LIN {X 0,Y 362.115,Z 224.377,A -85,B 0,C 180,E1 -12966.688,E2 -12966.688} C_VEL
LIN {X 0,Y 361.993,Z 224.393,A -85,B 0,C 180,E1 -12970.064,E2 -12970.064} C_VEL
LIN {X 0,Y 361.96,Z 224.393,A -85,B 0,C 180,E1 -12973.9,E2 -12973.9} C_VEL
LIN {X 0,Y 361.917,Z 224.398,A -85,B 0,C 180,E1 -12977.933,E2 -12977.933} C_VEL
LIN {X 0,Y 361.826,Z 224.413,A -85,B 0,C 180,E1 -12981.657,E2 -12981.657} C_VEL
LIN {X 0,Y 361.893,Z 224.405,A -85,B 0,C 180,E1 -12985.293,E2 -12985.293} C_VEL
LIN {X 0,Y 361.875,Z 224.406,A -85,B 0,C 180,E1 -12987.782,E2 -12987.782} C_VEL
LIN {X 0,Y 361.805,Z 224.415,A -85,B 0,C 180,E1 -12991.633,E2 -12991.633} C_VEL
LIN {X 0,Y 361.847,Z 224.405,A -85,B 0,C 180,E1 -12995.348,E2 -12995.348} C_VEL
LIN {X 0,Y 361.839,Z 224.413,A -85,B 0,C 180,E1 -12999.028,E2 -12999.028} C_VEL
LIN {X 0,Y 361.814,Z 224.411,A -85,B 0,C 180,E1 -13002.833,E2 -13002.833} C_VEL
LIN {X 0,Y 361.798,Z 224.416,A -85,B 0,C 180,E1 -13005.95,E2 -13005.95} C_VEL
LIN {X 0,Y 361.818,Z 224.414,A -85,B 0,C 180,E1 -13009.248,E2 -13009.248} C_VEL
LIN {X 0,Y 361.849,Z 224.412,A -85,B 0,C 180,E1 -13012.781,E2 -13012.781} C_VEL
LIN {X 0,Y 361.843,Z 224.414,A -85,B 0,C 180,E1 -13015.723,E2 -13015.723} C_VEL
LIN {X 0,Y 361.874,Z 224.521,A -85,B 0,C 180,E1 -13018.682,E2 -13018.682} C_VEL
LIN {X 0,Y 364.574,Z 235.414,A -85,B 0,C 180,E1 -13021.505,E2 -13021.505} C_VEL
LIN {X 0,Y 366.434,Z 244.952,A -85,B 0,C 180,E1 -13023.827,E2 -13023.827} C_VEL
LIN {X 0,Y 365.869,Z 253.146,A -85,B 0,C 180,E1 -13025.61,E2 -13025.61} C_VEL
LIN {X 0,Y 365.188,Z 259.855,A -85,B 0,C 180,E1 -13027.036,E2 -13027.036} C_VEL
LIN {X 0,Y 369.695,Z 284.03,A -85,B 0,C 180,E1 -13027.985,E2 -13027.985} C_VEL
LIN {X 0,Y 371.444,Z 298.142,A -85,B 0,C 180,E1 -13028.456,E2 -13028.456} C_VEL
LIN {X 0,Y 369.762,Z 370.004,A -85,B 0,C 180,E1 -13030.068,E2 -13030.068} C_VEL
LIN {X 0,Y 368.841,Z 384.089,A -85,B 0,C 180,E1 -13030.596,E2 -13030.596} C_VEL
LIN {X 0,Y 367.944,Z 396.187,A -85,B 0,C 180,E1 -13031.271,E2 -13031.271} C_VEL
LIN {X 0,Y 366.76,Z 407.982,A -85,B 0,C 180,E1 -13032.148,E2 -13032.148} C_VEL
LIN {X 0,Y 365.523,Z 419.416,A -85,B 0,C 180,E1 -13033.239,E2 -13033.239} C_VEL
LIN {X 0,Y 364.456,Z 428.714,A -85,B 0,C 180,E1 -13034.339,E2 -13034.339} C_VEL
LIN {X 0,Y 363.368,Z 438.309,A -85,B 0,C 180,E1 -13035.725,E2 -13035.725} C_VEL
LIN {X 0,Y 362.358,Z 447.58,A -85,B 0,C 180,E1 -13037.398,E2 -13037.398} C_VEL
LIN {X 0,Y 361.445,Z 455.08,A -85,B 0,C 180,E1 -13039.073,E2 -13039.073} C_VEL
LIN {X 0,Y 360.84,Z 461.992,A -85,B 0,C 180,E1 -13041.037,E2 -13041.037} C_VEL
LIN {X 0,Y 360.513,Z 466.581,A -85,B 0,C 180,E1 -13042.721,E2 -13042.721} C_VEL
LIN {X 0,Y 360.356,Z 470.071,A -85,B 0,C 180,E1 -13044.404,E2 -13044.404} C_VEL
LIN {X 0,Y 360.363,Z 471.821,A -85,B 0,C 180,E1 -13045.526,E2 -13045.526} C_VEL
LIN {X 0,Y 360.325,Z 473.156,A -85,B 0,C 180,E1 -13046.646,E2 -13046.646} C_VEL
LIN {X 0,Y 360.352,Z 474.073,A -85,B 0,C 180,E1 -13047.765,E2 -13047.765} C_VEL
LIN {X 0,Y 360.455,Z 474.543,A -85,B 0,C 180,E1 -13048.883,E2 -13048.883} C_VEL
LIN {X 0,Y 360.48,Z 474.608,A -85,B 0,C 180,E1 -13050,E2 -13050} C_VEL
LIN {X 0,Y 360.476,Z 474.272,A -85,B 0,C 180,E1 -13051.117,E2 -13051.117} C_VEL
LIN {X 0,Y 360.385,Z 473.507,A -85,B 0,C 180,E1 -13052.235,E2 -13052.235} C_VEL
LIN {X 0,Y 360.332,Z 472.287,A -85,B 0,C 180,E1 -13053.354,E2 -13053.354} C_VEL
LIN {X 0,Y 360.401,Z 469.667,A -85,B 0,C 180,E1 -13055.034,E2 -13055.034} C_VEL
LIN {X 0,Y 360.498,Z 465.984,A -85,B 0,C 180,E1 -13056.717,E2 -13056.717} C_VEL
LIN {X 0,Y 360.705,Z 461.141,A -85,B 0,C 180,E1 -13058.402,E2 -13058.402} C_VEL
LIN {X 0,Y 361.086,Z 454.997,A -85,B 0,C 180,E1 -13060.087,E2 -13060.087} C_VEL
LIN {X 0,Y 361.721,Z 447.337,A -85,B 0,C 180,E1 -13061.77,E2 -13061.77} C_VEL
LIN {X 0,Y 362.371,Z 439.494,A -85,B 0,C 180,E1 -13063.171,E2 -13063.171} C_VEL
LIN {X 0,Y 363.255,Z 429.911,A -85,B 0,C 180,E1 -13064.565,E2 -13064.565} C_VEL
LIN {X 0,Y 364.119,Z 419.27,A -85,B 0,C 180,E1 -13065.819,E2 -13065.819} C_VEL
LIN {X 0,Y 365.169,Z 407.451,A -85,B 0,C 180,E1 -13066.921,E2 -13066.921} C_VEL
LIN {X 0,Y 366.069,Z 394.843,A -85,B 0,C 180,E1 -13067.815,E2 -13067.815} C_VEL
LIN {X 0,Y 366.962,Z 381.699,A -85,B 0,C 180,E1 -13068.492,E2 -13068.492} C_VEL
LIN {X 0,Y 367.494,Z 368.498,A -85,B 0,C 180,E1 -13068.934,E2 -13068.934} C_VEL
LIN {X 0,Y 368.7,Z 295.929,A -85,B 0,C 180,E1 -13070.5,E2 -13070.5} C_VEL
LIN {X 0,Y 364.06,Z 262.327,A -85,B 0,C 180,E1 -13071.515,E2 -13071.515} C_VEL
LIN {X 0,Y 365.707,Z 244.487,A -85,B 0,C 180,E1 -13075.414,E2 -13075.414} C_VEL
LIN {X 0,Y 365.019,Z 239.454,A -85,B 0,C 180,E1 -13076.59,E2 -13076.59} C_VEL
LIN {X 0,Y 362.715,Z 228.266,A -85,B 0,C 180,E1 -13079.316,E2 -13079.316} C_VEL
LIN {X 0,Y 361.904,Z 224.406,A -85,B 0,C 180,E1 -13080.321,E2 -13080.321} C_VEL
LIN {X 0,Y 361.842,Z 224.412,A -85,B 0,C 180,E1 -13084.277,E2 -13084.277} C_VEL
LIN {X 0,Y 361.849,Z 224.409,A -85,B 0,C 180,E1 -13087.219,E2 -13087.219} C_VEL
LIN {X 0,Y 361.817,Z 224.412,A -85,B 0,C 180,E1 -13090.751,E2 -13090.751} C_VEL
LIN {X 0,Y 361.796,Z 224.416,A -85,B 0,C 180,E1 -13094.365,E2 -13094.365} C_VEL
LIN {X 0,Y 361.813,Z 224.417,A -85,B 0,C 180,E1 -13097.565,E2 -13097.565} C_VEL
LIN {X 0,Y 361.839,Z 224.41,A -85,B 0,C 180,E1 -13100.971,E2 -13100.971} C_VEL
LIN {X 0,Y 361.846,Z 224.408,A -85,B 0,C 180,E1 -13104.652,E2 -13104.652} C_VEL
LIN {X 0,Y 361.804,Z 224.414,A -85,B 0,C 180,E1 -13108.367,E2 -13108.367} C_VEL
LIN {X 0,Y 361.874,Z 224.405,A -85,B 0,C 180,E1 -13112.218,E2 -13112.218} C_VEL
LIN {X 0,Y 361.892,Z 224.403,A -85,B 0,C 180,E1 -13114.707,E2 -13114.707} C_VEL
LIN {X 0,Y 361.824,Z 224.411,A -85,B 0,C 180,E1 -13118.342,E2 -13118.342} C_VEL
LIN {X 0,Y 361.882,Z 224.404,A -85,B 0,C 180,E1 -13122.083,E2 -13122.083} C_VEL
LIN {X 0,Y 361.922,Z 224.404,A -85,B 0,C 180,E1 -13125.378,E2 -13125.378} C_VEL
LIN {X 0,Y 361.934,Z 224.4,A -85,B 0,C 180,E1 -13128.803,E2 -13128.803} C_VEL
LIN {X 0,Y 362.072,Z 224.38,A -85,B 0,C 180,E1 -13132.19,E2 -13132.19} C_VEL
LIN {X 0,Y 362.067,Z 224.382,A -85,B 0,C 180,E1 -13134.43,E2 -13134.43} C_VEL
LIN {X 0,Y 362.233,Z 224.36,A -85,B 0,C 180,E1 -13137.776,E2 -13137.776} C_VEL
LIN {X 0,Y 362.34,Z 224.347,A -85,B 0,C 180,E1 -13140,E2 -13140} C_VEL
LIN {X 0,Y 362.234,Z 224.361,A -85,B 0,C 180,E1 -13142.223,E2 -13142.223} C_VEL
LIN {X 0,Y 362.128,Z 224.378,A -85,B 0,C 180,E1 -13146.712,E2 -13146.712} C_VEL
LIN {X 0,Y 361.991,Z 224.391,A -85,B 0,C 180,E1 -13150.063,E2 -13150.063} C_VEL
LIN {X 0,Y 361.958,Z 224.395,A -85,B 0,C 180,E1 -13153.899,E2 -13153.899} C_VEL
LIN {X 0,Y 361.93,Z 224.399,A -85,B 0,C 180,E1 -13157.94,E2 -13157.94} C_VEL
LIN {X 0,Y 361.897,Z 224.402,A -85,B 0,C 180,E1 -13161.652,E2 -13161.652} C_VEL
LIN {X 0,Y 361.895,Z 224.402,A -85,B 0,C 180,E1 -13165.292,E2 -13165.292} C_VEL
LIN {X 0,Y 361.884,Z 224.405,A -85,B 0,C 180,E1 -13167.781,E2 -13167.781} C_VEL
LIN {X 0,Y 361.815,Z 224.412,A -85,B 0,C 180,E1 -13171.287,E2 -13171.287} C_VEL
LIN {X 0,Y 361.823,Z 224.418,A -85,B 0,C 180,E1 -13174.283,E2 -13174.283} C_VEL
LIN {X 0,Y 361.836,Z 224.41,A -85,B 0,C 180,E1 -13177.226,E2 -13177.226} C_VEL
LIN {X 0,Y 361.881,Z 224.405,A -85,B 0,C 180,E1 -13180.771,E2 -13180.771} C_VEL
LIN {X 0,Y 361.877,Z 224.408,A -85,B 0,C 180,E1 -13184.359,E2 -13184.359} C_VEL
LIN {X 0,Y 361.821,Z 224.413,A -85,B 0,C 180,E1 -13187.57,E2 -13187.57} C_VEL
LIN {X 0,Y 361.854,Z 224.407,A -85,B 0,C 180,E1 -13190.976,E2 -13190.976} C_VEL
LIN {X 0,Y 361.858,Z 224.407,A -85,B 0,C 180,E1 -13194.658,E2 -13194.658} C_VEL
LIN {X 0,Y 361.824,Z 224.412,A -85,B 0,C 180,E1 -13198.373,E2 -13198.373} C_VEL
LIN {X 0,Y 361.89,Z 224.403,A -85,B 0,C 180,E1 -13200.958,E2 -13200.958} C_VEL
LIN {X 0,Y 361.944,Z 224.4,A -85,B 0,C 180,E1 -13203.478,E2 -13203.478} C_VEL
LIN {X 0,Y 361.882,Z 224.406,A -85,B 0,C 180,E1 -13207.147,E2 -13207.147} C_VEL
LIN {X 0,Y 361.915,Z 224.4,A -85,B 0,C 180,E1 -13210.726,E2 -13210.726} C_VEL
LIN {X 0,Y 361.941,Z 224.397,A -85,B 0,C 180,E1 -13214.228,E2 -13214.228} C_VEL
LIN {X 0,Y 361.995,Z 224.39,A -85,B 0,C 180,E1 -13216.529,E2 -13216.529} C_VEL
LIN {X 0,Y 362.028,Z 224.387,A -85,B 0,C 180,E1 -13219.939,E2 -13219.939} C_VEL
LIN {X 0,Y 362.158,Z 224.376,A -85,B 0,C 180,E1 -13223.314,E2 -13223.314} C_VEL
LIN {X 0,Y 362.281,Z 224.356,A -85,B 0,C 180,E1 -13227.777,E2 -13227.777} C_VEL
LIN {X 0,Y 362.425,Z 224.337,A -85,B 0,C 180,E1 -13230,E2 -13230} C_VEL
LIN {X 0,Y 362.281,Z 224.354,A -85,B 0,C 180,E1 -13232.223,E2 -13232.223} C_VEL
LIN {X 0,Y 362.151,Z 224.373,A -85,B 0,C 180,E1 -13236.686,E2 -13236.686} C_VEL
LIN {X 0,Y 362.029,Z 224.386,A -85,B 0,C 180,E1 -13240.061,E2 -13240.061} C_VEL
LIN {X 0,Y 361.994,Z 224.39,A -85,B 0,C 180,E1 -13243.897,E2 -13243.897} C_VEL
LIN {X 0,Y 361.962,Z 224.394,A -85,B 0,C 180,E1 -13247.937,E2 -13247.937} C_VEL
LIN {X 0,Y 361.855,Z 224.407,A -85,B 0,C 180,E1 -13251.653,E2 -13251.653} C_VEL
LIN {X 0,Y 361.917,Z 224.405,A -85,B 0,C 180,E1 -13255.288,E2 -13255.288} C_VEL
LIN {X 0,Y 361.972,Z 224.536,A -85,B 0,C 180,E1 -13256.937,E2 -13256.937} C_VEL
LIN {X 0,Y 363.133,Z 230.494,A -85,B 0,C 180,E1 -13258.538,E2 -13258.538} C_VEL
LIN {X 0,Y 367.197,Z 242.914,A -85,B 0,C 180,E1 -13259.039,E2 -13259.039} C_VEL
LIN {X 0,Y 369.399,Z 254.487,A -85,B 0,C 180,E1 -13259.415,E2 -13259.415} C_VEL
LIN {X 0,Y 367.623,Z 338.548,A -85,B 0,C 180,E1 -13261.232,E2 -13261.232} C_VEL
LIN {X 0,Y 367.262,Z 348.263,A -85,B 0,C 180,E1 -13261.578,E2 -13261.578} C_VEL
LIN {X 0,Y 366.329,Z 353.922,A -85,B 0,C 180,E1 -13261.81,E2 -13261.81} C_VEL
LIN {X 0,Y 363.1,Z 362.978,A -85,B 0,C 180,E1 -13262.204,E2 -13262.204} C_VEL
LIN {X 0,Y 359.835,Z 371.762,A -85,B 0,C 180,E1 -13262.714,E2 -13262.714} C_VEL
LIN {X 0,Y 358.859,Z 376.971,A -85,B 0,C 180,E1 -13263.125,E2 -13263.125} C_VEL
LIN {X 0,Y 357.964,Z 387.984,A -85,B 0,C 180,E1 -13264.214,E2 -13264.214} C_VEL
LIN {X 0,Y 357.088,Z 398.297,A -85,B 0,C 180,E1 -13265.488,E2 -13265.488} C_VEL
LIN {X 0,Y 356.157,Z 408.096,A -85,B 0,C 180,E1 -13266.998,E2 -13266.998} C_VEL
LIN {X 0,Y 355.399,Z 416.152,A -85,B 0,C 180,E1 -13268.523,E2 -13268.523} C_VEL
LIN {X 0,Y 354.695,Z 423.012,A -85,B 0,C 180,E1 -13270.113,E2 -13270.113} C_VEL
LIN {X 0,Y 354.165,Z 428.666,A -85,B 0,C 180,E1 -13271.734,E2 -13271.734} C_VEL
LIN {X 0,Y 353.836,Z 433.362,A -85,B 0,C 180,E1 -13273.432,E2 -13273.432} C_VEL
LIN {X 0,Y 353.551,Z 436.816,A -85,B 0,C 180,E1 -13275.061,E2 -13275.061} C_VEL
LIN {X 0,Y 353.408,Z 438.217,A -85,B 0,C 180,E1 -13275.892,E2 -13275.892} C_VEL
LIN {X 0,Y 353.225,Z 440.195,A -85,B 0,C 180,E1 -13277.431,E2 -13277.431} C_VEL
LIN {X 0,Y 353.132,Z 441.501,A -85,B 0,C 180,E1 -13279.129,E2 -13279.129} C_VEL
LIN {X 0,Y 353.142,Z 441.899,A -85,B 0,C 180,E1 -13280.902,E2 -13280.902} C_VEL
LIN {X 0,Y 353.278,Z 441.286,A -85,B 0,C 180,E1 -13282.718,E2 -13282.718} C_VEL
LIN {X 0,Y 353.577,Z 439.303,A -85,B 0,C 180,E1 -13284.801,E2 -13284.801} C_VEL
LIN {X 0,Y 353.938,Z 436.632,A -85,B 0,C 180,E1 -13286.5,E2 -13286.5} C_VEL
LIN {X 0,Y 354.553,Z 432.301,A -85,B 0,C 180,E1 -13288.458,E2 -13288.458} C_VEL
LIN {X 0,Y 355.312,Z 426.61,A -85,B 0,C 180,E1 -13290.364,E2 -13290.364} C_VEL
LIN {X 0,Y 356.242,Z 419.66,A -85,B 0,C 180,E1 -13292.169,E2 -13292.169} C_VEL
LIN {X 0,Y 357.296,Z 412.146,A -85,B 0,C 180,E1 -13293.732,E2 -13293.732} C_VEL
LIN {X 0,Y 358.362,Z 403.424,A -85,B 0,C 180,E1 -13295.217,E2 -13295.217} C_VEL
LIN {X 0,Y 359.516,Z 393.604,A -85,B 0,C 180,E1 -13296.565,E2 -13296.565} C_VEL
LIN {X 0,Y 360.868,Z 381.992,A -85,B 0,C 180,E1 -13297.832,E2 -13297.832} C_VEL
LIN {X 0,Y 361.902,Z 370.101,A -85,B 0,C 180,E1 -13298.85,E2 -13298.85} C_VEL
LIN {X 0,Y 362.86,Z 357.252,A -85,B 0,C 180,E1 -13299.671,E2 -13299.671} C_VEL
LIN {X 0,Y 363.499,Z 344.303,A -85,B 0,C 180,E1 -13300.261,E2 -13300.261} C_VEL
LIN {X 0,Y 363.987,Z 329.813,A -85,B 0,C 180,E1 -13300.655,E2 -13300.655} C_VEL
LIN {X 0,Y 365.902,Z 256.319,A -85,B 0,C 180,E1 -13302.319,E2 -13302.319} C_VEL
LIN {X 0,Y 364.36,Z 250.049,A -85,B 0,C 180,E1 -13302.604,E2 -13302.604} C_VEL
LIN {X 0,Y 358.053,Z 235.223,A -85,B 0,C 180,E1 -13303.523,E2 -13303.523} C_VEL
LIN {X 0,Y 356.561,Z 231.883,A -85,B 0,C 180,E1 -13303.784,E2 -13303.784} C_VEL
LIN {X 0,Y 354.918,Z 225.281,A -85,B 0,C 180,E1 -13305.625,E2 -13305.625} C_VEL
LIN {X 0,Y 354.94,Z 225.278,A -85,B 0,C 180,E1 -13309.735,E2 -13309.735} C_VEL
LIN {X 0,Y 355.09,Z 225.255,A -85,B 0,C 180,E1 -13313.18,E2 -13313.18} C_VEL
LIN {X 0,Y 355.199,Z 225.241,A -85,B 0,C 180,E1 -13317.732,E2 -13317.732} C_VEL
LIN {X 0,Y 355.311,Z 225.226,A -85,B 0,C 180,E1 -13320,E2 -13320} C_VEL
LIN {X 0,Y 355.198,Z 225.24,A -85,B 0,C 180,E1 -13322.268,E2 -13322.268} C_VEL
LIN {X 0,Y 355.079,Z 225.255,A -85,B 0,C 180,E1 -13326.821,E2 -13326.821} C_VEL
LIN {X 0,Y 354.94,Z 225.272,A -85,B 0,C 180,E1 -13330.266,E2 -13330.266} C_VEL
LIN {X 0,Y 354.905,Z 225.272,A -85,B 0,C 180,E1 -13334.019,E2 -13334.019} C_VEL
LIN {X 0,Y 354.876,Z 225.276,A -85,B 0,C 180,E1 -13338.105,E2 -13338.105} C_VEL
LIN {X 0,Y 354.781,Z 225.292,A -85,B 0,C 180,E1 -13342.11,E2 -13342.11} C_VEL
LIN {X 0,Y 354.865,Z 225.28,A -85,B 0,C 180,E1 -13345.831,E2 -13345.831} C_VEL
LIN {X 0,Y 354.773,Z 225.286,A -85,B 0,C 180,E1 -13349.686,E2 -13349.686} C_VEL
LIN {X 0,Y 354.789,Z 225.289,A -85,B 0,C 180,E1 -13353.687,E2 -13353.687} C_VEL
LIN {X 0,Y 354.771,Z 225.294,A -85,B 0,C 180,E1 -13356.463,E2 -13356.463} C_VEL
LIN {X 0,Y 354.803,Z 225.289,A -85,B 0,C 180,E1 -13359.427,E2 -13359.427} C_VEL
LIN {X 0,Y 354.766,Z 225.289,A -85,B 0,C 180,E1 -13362.87,E2 -13362.87} C_VEL
LIN {X 0,Y 354.748,Z 225.295,A -85,B 0,C 180,E1 -13366.107,E2 -13366.107} C_VEL
LIN {X 0,Y 354.771,Z 225.292,A -85,B 0,C 180,E1 -13369.182,E2 -13369.182} C_VEL
LIN {X 0,Y 354.793,Z 225.293,A -85,B 0,C 180,E1 -13372.406,E2 -13372.406} C_VEL
LIN {X 0,Y 354.8,Z 225.288,A -85,B 0,C 180,E1 -13374.944,E2 -13374.944} C_VEL
LIN {X 0,Y 354.811,Z 225.417,A -85,B 0,C 180,E1 -13378.145,E2 -13378.145} C_VEL
LIN {X 0,Y 357.708,Z 236.939,A -85,B 0,C 180,E1 -13381.229,E2 -13381.229} C_VEL
LIN {X 0,Y 359.523,Z 246.075,A -85,B 0,C 180,E1 -13383.517,E2 -13383.517} C_VEL
LIN {X 0,Y 359.46,Z 250.516,A -85,B 0,C 180,E1 -13384.527,E2 -13384.527} C_VEL
LIN {X 0,Y 358.516,Z 259.669,A -85,B 0,C 180,E1 -13386.482,E2 -13386.482} C_VEL
LIN {X 0,Y 362.754,Z 281.64,A -85,B 0,C 180,E1 -13387.395,E2 -13387.395} C_VEL
LIN {X 0,Y 365.014,Z 298.796,A -85,B 0,C 180,E1 -13387.996,E2 -13387.996} C_VEL
LIN {X 0,Y 363.234,Z 369.682,A -85,B 0,C 180,E1 -13389.621,E2 -13389.621} C_VEL
LIN {X 0,Y 362.307,Z 383.682,A -85,B 0,C 180,E1 -13390.158,E2 -13390.158} C_VEL
LIN {X 0,Y 361.326,Z 395.747,A -85,B 0,C 180,E1 -13390.841,E2 -13390.841} C_VEL
LIN {X 0,Y 360.209,Z 406.735,A -85,B 0,C 180,E1 -13391.665,E2 -13391.665} C_VEL
LIN {X 0,Y 358.871,Z 418.31,A -85,B 0,C 180,E1 -13392.772,E2 -13392.772} C_VEL
LIN {X 0,Y 357.621,Z 428.82,A -85,B 0,C 180,E1 -13394.032,E2 -13394.032} C_VEL
LIN {X 0,Y 356.484,Z 438.319,A -85,B 0,C 180,E1 -13395.443,E2 -13395.443} C_VEL
LIN {X 0,Y 355.399,Z 447.532,A -85,B 0,C 180,E1 -13397.147,E2 -13397.147} C_VEL
LIN {X 0,Y 354.422,Z 454.987,A -85,B 0,C 180,E1 -13398.854,E2 -13398.854} C_VEL
LIN {X 0,Y 353.95,Z 460.048,A -85,B 0,C 180,E1 -13400.284,E2 -13400.284} C_VEL
LIN {X 0,Y 353.545,Z 464.985,A -85,B 0,C 180,E1 -13402.002,E2 -13402.002} C_VEL
LIN {X 0,Y 353.297,Z 469.445,A -85,B 0,C 180,E1 -13404.064,E2 -13404.064} C_VEL
LIN {X 0,Y 353.273,Z 471.556,A -85,B 0,C 180,E1 -13405.436,E2 -13405.436} C_VEL
LIN {X 0,Y 353.245,Z 472.878,A -85,B 0,C 180,E1 -13406.578,E2 -13406.578} C_VEL
LIN {X 0,Y 353.253,Z 473.765,A -85,B 0,C 180,E1 -13407.72,E2 -13407.72} C_VEL
LIN {X 0,Y 353.357,Z 474.218,A -85,B 0,C 180,E1 -13408.86,E2 -13408.86} C_VEL
LIN {X 0,Y 353.399,Z 474.269,A -85,B 0,C 180,E1 -13410,E2 -13410} C_VEL
LIN {X 0,Y 353.378,Z 473.915,A -85,B 0,C 180,E1 -13411.139,E2 -13411.139} C_VEL
LIN {X 0,Y 353.288,Z 473.116,A -85,B 0,C 180,E1 -13412.28,E2 -13412.28} C_VEL
LIN {X 0,Y 353.253,Z 471.879,A -85,B 0,C 180,E1 -13413.421,E2 -13413.421} C_VEL
LIN {X 0,Y 353.302,Z 469.218,A -85,B 0,C 180,E1 -13415.135,E2 -13415.135} C_VEL
LIN {X 0,Y 353.417,Z 465.492,A -85,B 0,C 180,E1 -13416.852,E2 -13416.852} C_VEL
LIN {X 0,Y 353.647,Z 460.602,A -85,B 0,C 180,E1 -13418.571,E2 -13418.571} C_VEL
LIN {X 0,Y 354.046,Z 454.404,A -85,B 0,C 180,E1 -13420.29,E2 -13420.29} C_VEL
LIN {X 0,Y 354.73,Z 446.681,A -85,B 0,C 180,E1 -13422.005,E2 -13422.005} C_VEL
LIN {X 0,Y 355.423,Z 438.753,A -85,B 0,C 180,E1 -13423.433,E2 -13423.433} C_VEL
LIN {X 0,Y 356.468,Z 428.191,A -85,B 0,C 180,E1 -13424.967,E2 -13424.967} C_VEL
LIN {X 0,Y 357.34,Z 416.984,A -85,B 0,C 180,E1 -13426.274,E2 -13426.274} C_VEL
LIN {X 0,Y 358.453,Z 404.493,A -85,B 0,C 180,E1 -13427.395,E2 -13427.395} C_VEL
LIN {X 0,Y 359.4,Z 392.315,A -85,B 0,C 180,E1 -13428.231,E2 -13428.231} C_VEL
LIN {X 0,Y 360.202,Z 378.807,A -85,B 0,C 180,E1 -13428.888,E2 -13428.888} C_VEL
LIN {X 0,Y 360.725,Z 365.466,A -85,B 0,C 180,E1 -13429.303,E2 -13429.303} C_VEL
LIN {X 0,Y 361.926,Z 296.685,A -85,B 0,C 180,E1 -13430.812,E2 -13430.812} C_VEL
LIN {X 0,Y 357.159,Z 262.03,A -85,B 0,C 180,E1 -13431.881,E2 -13431.881} C_VEL
LIN {X 0,Y 358.729,Z 245.661,A -85,B 0,C 180,E1 -13435.529,E2 -13435.529} C_VEL
LIN {X 0,Y 358.222,Z 241.554,A -85,B 0,C 180,E1 -13436.507,E2 -13436.507} C_VEL
LIN {X 0,Y 355.827,Z 229.809,A -85,B 0,C 180,E1 -13439.414,E2 -13439.414} C_VEL
LIN {X 0,Y 354.838,Z 225.285,A -85,B 0,C 180,E1 -13440.578,E2 -13440.578} C_VEL
LIN {X 0,Y 354.796,Z 225.29,A -85,B 0,C 180,E1 -13443.699,E2 -13443.699} C_VEL
LIN {X 0,Y 354.784,Z 225.29,A -85,B 0,C 180,E1 -13446.456,E2 -13446.456} C_VEL
LIN {X 0,Y 354.81,Z 225.287,A -85,B 0,C 180,E1 -13449.42,E2 -13449.42} C_VEL
LIN {X 0,Y 354.77,Z 225.29,A -85,B 0,C 180,E1 -13452.863,E2 -13452.863} C_VEL
LIN {X 0,Y 354.745,Z 225.296,A -85,B 0,C 180,E1 -13456.1,E2 -13456.1} C_VEL
LIN {X 0,Y 354.763,Z 225.292,A -85,B 0,C 180,E1 -13459.175,E2 -13459.175} C_VEL
LIN {X 0,Y 354.78,Z 225.289,A -85,B 0,C 180,E1 -13462.4,E2 -13462.4} C_VEL
LIN {X 0,Y 354.784,Z 225.289,A -85,B 0,C 180,E1 -13464.937,E2 -13464.937} C_VEL
LIN {X 0,Y 354.76,Z 225.291,A -85,B 0,C 180,E1 -13468.403,E2 -13468.403} C_VEL
LIN {X 0,Y 354.798,Z 225.291,A -85,B 0,C 180,E1 -13471.614,E2 -13471.614} C_VEL
LIN {X 0,Y 354.864,Z 225.279,A -85,B 0,C 180,E1 -13474.169,E2 -13474.169} C_VEL
LIN {X 0,Y 354.779,Z 225.29,A -85,B 0,C 180,E1 -13477.89,E2 -13477.89} C_VEL
LIN {X 0,Y 354.853,Z 225.28,A -85,B 0,C 180,E1 -13481.906,E2 -13481.906} C_VEL
LIN {X 0,Y 354.904,Z 225.273,A -85,B 0,C 180,E1 -13485.981,E2 -13485.981} C_VEL
LIN {X 0,Y 354.939,Z 225.27,A -85,B 0,C 180,E1 -13489.734,E2 -13489.734} C_VEL
LIN {X 0,Y 355.078,Z 225.257,A -85,B 0,C 180,E1 -13493.179,E2 -13493.179} C_VEL
LIN {X 0,Y 355.197,Z 225.237,A -85,B 0,C 180,E1 -13497.732,E2 -13497.732} C_VEL
LIN {X 0,Y 355.291,Z 225.225,A -85,B 0,C 180,E1 -13500,E2 -13500} C_VEL
LIN {X 0,Y 355.198,Z 225.237,A -85,B 0,C 180,E1 -13502.268,E2 -13502.268} C_VEL
LIN {X 0,Y 355.093,Z 225.256,A -85,B 0,C 180,E1 -13506.82,E2 -13506.82} C_VEL
LIN {X 0,Y 354.939,Z 225.271,A -85,B 0,C 180,E1 -13510.265,E2 -13510.265} C_VEL
LIN {X 0,Y 354.903,Z 225.274,A -85,B 0,C 180,E1 -13514.019,E2 -13514.019} C_VEL
LIN {X 0,Y 354.886,Z 225.277,A -85,B 0,C 180,E1 -13518.11,E2 -13518.11} C_VEL
LIN {X 0,Y 354.857,Z 225.281,A -85,B 0,C 180,E1 -13522.104,E2 -13522.104} C_VEL
LIN {X 0,Y 354.865,Z 225.279,A -85,B 0,C 180,E1 -13525.83,E2 -13525.83} C_VEL
LIN {X 0,Y 354.822,Z 225.284,A -85,B 0,C 180,E1 -13529.681,E2 -13529.681} C_VEL
LIN {X 0,Y 354.777,Z 225.29,A -85,B 0,C 180,E1 -13533.705,E2 -13533.705} C_VEL
LIN {X 0,Y 354.77,Z 225.294,A -85,B 0,C 180,E1 -13536.462,E2 -13536.462} C_VEL
LIN {X 0,Y 354.799,Z 225.287,A -85,B 0,C 180,E1 -13539.426,E2 -13539.426} C_VEL
LIN {X 0,Y 354.811,Z 225.285,A -85,B 0,C 180,E1 -13542.878,E2 -13542.878} C_VEL
LIN {X 0,Y 354.76,Z 225.297,A -85,B 0,C 180,E1 -13546.109,E2 -13546.109} C_VEL
LIN {X 0,Y 354.799,Z 225.286,A -85,B 0,C 180,E1 -13549.186,E2 -13549.186} C_VEL
LIN {X 0,Y 354.791,Z 225.289,A -85,B 0,C 180,E1 -13552.405,E2 -13552.405} C_VEL
LIN {X 0,Y 354.796,Z 225.287,A -85,B 0,C 180,E1 -13554.944,E2 -13554.944} C_VEL
LIN {X 0,Y 354.78,Z 225.29,A -85,B 0,C 180,E1 -13558.408,E2 -13558.408} C_VEL
LIN {X 0,Y 354.842,Z 225.286,A -85,B 0,C 180,E1 -13561.622,E2 -13561.622} C_VEL
LIN {X 0,Y 354.889,Z 225.277,A -85,B 0,C 180,E1 -13564.175,E2 -13564.175} C_VEL
LIN {X 0,Y 354.827,Z 225.286,A -85,B 0,C 180,E1 -13567.896,E2 -13567.896} C_VEL
LIN {X 0,Y 354.917,Z 225.274,A -85,B 0,C 180,E1 -13571.893,E2 -13571.893} C_VEL
LIN {X 0,Y 354.938,Z 225.27,A -85,B 0,C 180,E1 -13575.983,E2 -13575.983} C_VEL
LIN {X 0,Y 354.975,Z 225.267,A -85,B 0,C 180,E1 -13579.737,E2 -13579.737} C_VEL
LIN {X 0,Y 355.123,Z 225.251,A -85,B 0,C 180,E1 -13583.181,E2 -13583.181} C_VEL
LIN {X 0,Y 355.244,Z 225.233,A -85,B 0,C 180,E1 -13587.733,E2 -13587.733} C_VEL
LIN {X 0,Y 355.395,Z 225.212,A -85,B 0,C 180,E1 -13590,E2 -13590} C_VEL
LIN {X 0,Y 355.244,Z 225.231,A -85,B 0,C 180,E1 -13592.267,E2 -13592.267} C_VEL
LIN {X 0,Y 355.116,Z 225.25,A -85,B 0,C 180,E1 -13596.819,E2 -13596.819} C_VEL
LIN {X 0,Y 354.975,Z 225.265,A -85,B 0,C 180,E1 -13600.263,E2 -13600.263} C_VEL
LIN {X 0,Y 354.939,Z 225.269,A -85,B 0,C 180,E1 -13604.017,E2 -13604.017} C_VEL
LIN {X 0,Y 354.917,Z 225.272,A -85,B 0,C 180,E1 -13608.107,E2 -13608.107} C_VEL
LIN {X 0,Y 354.809,Z 225.286,A -85,B 0,C 180,E1 -13612.105,E2 -13612.105} C_VEL
LIN {X 0,Y 354.898,Z 225.278,A -85,B 0,C 180,E1 -13615.824,E2 -13615.824} C_VEL
LIN {X 0,Y 354.955,Z 225.341,A -85,B 0,C 180,E1 -13616.664,E2 -13616.664} C_VEL
LIN {X 0,Y 355.999,Z 230.651,A -85,B 0,C 180,E1 -13618.145,E2 -13618.145} C_VEL
LIN {X 0,Y 360.627,Z 244.841,A -85,B 0,C 180,E1 -13618.738,E2 -13618.738} C_VEL
LIN {X 0,Y 362.633,Z 256.13,A -85,B 0,C 180,E1 -13619.107,E2 -13619.107} C_VEL
LIN {X 0,Y 360.79,Z 339.016,A -85,B 0,C 180,E1 -13620.937,E2 -13620.937} C_VEL
LIN {X 0,Y 360.218,Z 352.523,A -85,B 0,C 180,E1 -13621.468,E2 -13621.468} C_VEL
LIN {X 0,Y 359.641,Z 365.466,A -85,B 0,C 180,E1 -13622.227,E2 -13622.227} C_VEL
LIN {X 0,Y 358.859,Z 376.971,A -85,B 0,C 180,E1 -13623.125,E2 -13623.125} C_VEL
LIN {X 0,Y 357.867,Z 382.128,A -85,B 0,C 180,E1 -13623.577,E2 -13623.577} C_VEL
LIN {X 0,Y 354.458,Z 390.195,A -85,B 0,C 180,E1 -13624.334,E2 -13624.334} C_VEL
LIN {X 0,Y 350.943,Z 397.796,A -85,B 0,C 180,E1 -13625.189,E2 -13625.189} C_VEL
LIN {X 0,Y 349.775,Z 402.191,A -85,B 0,C 180,E1 -13625.796,E2 -13625.796} C_VEL
LIN {X 0,Y 348.799,Z 411.724,A -85,B 0,C 180,E1 -13627.411,E2 -13627.411} C_VEL
LIN {X 0,Y 348.071,Z 419.314,A -85,B 0,C 180,E1 -13629,E2 -13629} C_VEL
LIN {X 0,Y 347.385,Z 426.608,A -85,B 0,C 180,E1 -13630.899,E2 -13630.899} C_VEL
LIN {X 0,Y 346.952,Z 431.555,A -85,B 0,C 180,E1 -13632.532,E2 -13632.532} C_VEL
LIN {X 0,Y 346.64,Z 435.473,A -85,B 0,C 180,E1 -13634.175,E2 -13634.175} C_VEL
LIN {X 0,Y 346.453,Z 437.499,A -85,B 0,C 180,E1 -13635.228,E2 -13635.228} C_VEL
LIN {X 0,Y 346.158,Z 440.007,A -85,B 0,C 180,E1 -13636.955,E2 -13636.955} C_VEL
LIN {X 0,Y 346.067,Z 441.58,A -85,B 0,C 180,E1 -13638.705,E2 -13638.705} C_VEL
LIN {X 0,Y 346.057,Z 442.237,A -85,B 0,C 180,E1 -13640.982,E2 -13640.982} C_VEL
LIN {X 0,Y 346.188,Z 441.846,A -85,B 0,C 180,E1 -13642.481,E2 -13642.481} C_VEL
LIN {X 0,Y 346.369,Z 440.489,A -85,B 0,C 180,E1 -13644.246,E2 -13644.246} C_VEL
LIN {X 0,Y 346.78,Z 437.897,A -85,B 0,C 180,E1 -13646.185,E2 -13646.185} C_VEL
LIN {X 0,Y 347.433,Z 433.678,A -85,B 0,C 180,E1 -13648.269,E2 -13648.269} C_VEL
LIN {X 0,Y 348.184,Z 428.332,A -85,B 0,C 180,E1 -13650.21,E2 -13650.21} C_VEL
LIN {X 0,Y 349.111,Z 421.757,A -85,B 0,C 180,E1 -13652.063,E2 -13652.063} C_VEL
LIN {X 0,Y 350.331,Z 413.84,A -85,B 0,C 180,E1 -13653.811,E2 -13653.811} C_VEL
LIN {X 0,Y 351.562,Z 404.378,A -85,B 0,C 180,E1 -13655.493,E2 -13655.493} C_VEL
LIN {X 0,Y 352.75,Z 394.91,A -85,B 0,C 180,E1 -13656.845,E2 -13656.845} C_VEL
LIN {X 0,Y 354.046,Z 384.237,A -85,B 0,C 180,E1 -13658.061,E2 -13658.061} C_VEL
LIN {X 0,Y 355.224,Z 372.344,A -85,B 0,C 180,E1 -13659.138,E2 -13659.138} C_VEL
LIN {X 0,Y 356.169,Z 360.62,A -85,B 0,C 180,E1 -13659.95,E2 -13659.95} C_VEL
LIN {X 0,Y 356.914,Z 347.135,A -85,B 0,C 180,E1 -13660.622,E2 -13660.622} C_VEL
LIN {X 0,Y 357.447,Z 334.632,A -85,B 0,C 180,E1 -13661.018,E2 -13661.018} C_VEL
LIN {X 0,Y 359.621,Z 257.658,A -85,B 0,C 180,E1 -13662.803,E2 -13662.803} C_VEL
LIN {X 0,Y 358.087,Z 252.005,A -85,B 0,C 180,E1 -13663.081,E2 -13663.081} C_VEL
LIN {X 0,Y 352.134,Z 238.191,A -85,B 0,C 180,E1 -13663.98,E2 -13663.98} C_VEL
LIN {X 0,Y 349.43,Z 232.448,A -85,B 0,C 180,E1 -13664.406,E2 -13664.406} C_VEL
LIN {X 0,Y 347.887,Z 226.158,A -85,B 0,C 180,E1 -13666.269,E2 -13666.269} C_VEL
LIN {X 0,Y 347.891,Z 226.158,A -85,B 0,C 180,E1 -13669.525,E2 -13669.525} C_VEL
LIN {X 0,Y 348.055,Z 226.131,A -85,B 0,C 180,E1 -13673.042,E2 -13673.042} C_VEL
LIN {X 0,Y 348.162,Z 226.118,A -85,B 0,C 180,E1 -13677.687,E2 -13677.687} C_VEL
LIN {X 0,Y 348.263,Z 226.104,A -85,B 0,C 180,E1 -13680,E2 -13680} C_VEL
LIN {X 0,Y 348.161,Z 226.117,A -85,B 0,C 180,E1 -13682.314,E2 -13682.314} C_VEL
LIN {X 0,Y 348.047,Z 226.132,A -85,B 0,C 180,E1 -13686.959,E2 -13686.959} C_VEL
LIN {X 0,Y 347.891,Z 226.151,A -85,B 0,C 180,E1 -13690.476,E2 -13690.476} C_VEL
LIN {X 0,Y 347.864,Z 226.149,A -85,B 0,C 180,E1 -13694.152,E2 -13694.152} C_VEL
LIN {X 0,Y 347.81,Z 226.157,A -85,B 0,C 180,E1 -13698.269,E2 -13698.269} C_VEL
LIN {X 0,Y 347.733,Z 226.169,A -85,B 0,C 180,E1 -13701.627,E2 -13701.627} C_VEL
LIN {X 0,Y 347.779,Z 226.164,A -85,B 0,C 180,E1 -13705.111,E2 -13705.111} C_VEL
LIN {X 0,Y 347.771,Z 226.162,A -85,B 0,C 180,E1 -13707.698,E2 -13707.698} C_VEL
LIN {X 0,Y 347.713,Z 226.171,A -85,B 0,C 180,E1 -13711.703,E2 -13711.703} C_VEL
LIN {X 0,Y 347.718,Z 226.171,A -85,B 0,C 180,E1 -13714.467,E2 -13714.467} C_VEL
LIN {X 0,Y 347.747,Z 226.166,A -85,B 0,C 180,E1 -13717.991,E2 -13717.991} C_VEL
LIN {X 0,Y 347.728,Z 226.17,A -85,B 0,C 180,E1 -13721.834,E2 -13721.834} C_VEL
LIN {X 0,Y 347.685,Z 226.172,A -85,B 0,C 180,E1 -13725.031,E2 -13725.031} C_VEL
LIN {X 0,Y 347.734,Z 226.171,A -85,B 0,C 180,E1 -13728.401,E2 -13728.401} C_VEL
LIN {X 0,Y 347.759,Z 226.166,A -85,B 0,C 180,E1 -13732.015,E2 -13732.015} C_VEL
LIN {X 0,Y 347.734,Z 226.17,A -85,B 0,C 180,E1 -13735.539,E2 -13735.539} C_VEL
LIN {X 0,Y 347.744,Z 226.255,A -85,B 0,C 180,E1 -13737.563,E2 -13737.563} C_VEL
LIN {X 0,Y 350.581,Z 237.158,A -85,B 0,C 180,E1 -13740.588,E2 -13740.588} C_VEL
LIN {X 0,Y 352.693,Z 247.677,A -85,B 0,C 180,E1 -13743.306,E2 -13743.306} C_VEL
LIN {X 0,Y 352.656,Z 252.007,A -85,B 0,C 180,E1 -13744.316,E2 -13744.316} C_VEL
LIN {X 0,Y 351.858,Z 259.022,A -85,B 0,C 180,E1 -13745.874,E2 -13745.874} C_VEL
LIN {X 0,Y 356.092,Z 280.965,A -85,B 0,C 180,E1 -13746.831,E2 -13746.831} C_VEL
LIN {X 0,Y 358.554,Z 298.254,A -85,B 0,C 180,E1 -13747.482,E2 -13747.482} C_VEL
LIN {X 0,Y 357.054,Z 357.395,A -85,B 0,C 180,E1 -13748.848,E2 -13748.848} C_VEL
LIN {X 0,Y 356.54,Z 373.684,A -85,B 0,C 180,E1 -13749.296,E2 -13749.296} C_VEL
LIN {X 0,Y 355.426,Z 387.387,A -85,B 0,C 180,E1 -13749.908,E2 -13749.908} C_VEL
LIN {X 0,Y 354.242,Z 400.349,A -85,B 0,C 180,E1 -13750.744,E2 -13750.744} C_VEL
LIN {X 0,Y 352.952,Z 411.807,A -85,B 0,C 180,E1 -13751.725,E2 -13751.725} C_VEL
LIN {X 0,Y 351.488,Z 423.483,A -85,B 0,C 180,E1 -13752.999,E2 -13752.999} C_VEL
LIN {X 0,Y 350.177,Z 433.966,A -85,B 0,C 180,E1 -13754.442,E2 -13754.442} C_VEL
LIN {X 0,Y 349.024,Z 443.147,A -85,B 0,C 180,E1 -13756.019,E2 -13756.019} C_VEL
LIN {X 0,Y 347.902,Z 451.389,A -85,B 0,C 180,E1 -13757.755,E2 -13757.755} C_VEL
LIN {X 0,Y 347.147,Z 458.033,A -85,B 0,C 180,E1 -13759.503,E2 -13759.503} C_VEL
LIN {X 0,Y 346.629,Z 463.327,A -85,B 0,C 180,E1 -13761.254,E2 -13761.254} C_VEL
LIN {X 0,Y 346.322,Z 467.456,A -85,B 0,C 180,E1 -13763.007,E2 -13763.007} C_VEL
LIN {X 0,Y 346.202,Z 469.592,A -85,B 0,C 180,E1 -13764.175,E2 -13764.175} C_VEL
LIN {X 0,Y 346.169,Z 471.306,A -85,B 0,C 180,E1 -13765.342,E2 -13765.342} C_VEL
LIN {X 0,Y 346.166,Z 472.609,A -85,B 0,C 180,E1 -13766.508,E2 -13766.508} C_VEL
LIN {X 0,Y 346.159,Z 473.458,A -85,B 0,C 180,E1 -13767.673,E2 -13767.673} C_VEL
LIN {X 0,Y 346.259,Z 473.894,A -85,B 0,C 180,E1 -13768.837,E2 -13768.837} C_VEL
LIN {X 0,Y 346.32,Z 473.929,A -85,B 0,C 180,E1 -13770,E2 -13770} C_VEL
LIN {X 0,Y 346.281,Z 473.555,A -85,B 0,C 180,E1 -13771.163,E2 -13771.163} C_VEL
LIN {X 0,Y 346.191,Z 472.722,A -85,B 0,C 180,E1 -13772.327,E2 -13772.327} C_VEL
LIN {X 0,Y 346.176,Z 471.468,A -85,B 0,C 180,E1 -13773.491,E2 -13773.491} C_VEL
LIN {X 0,Y 346.21,Z 468.767,A -85,B 0,C 180,E1 -13775.241,E2 -13775.241} C_VEL
LIN {X 0,Y 346.341,Z 464.998,A -85,B 0,C 180,E1 -13776.992,E2 -13776.992} C_VEL
LIN {X 0,Y 346.571,Z 460.059,A -85,B 0,C 180,E1 -13778.747,E2 -13778.747} C_VEL
LIN {X 0,Y 346.988,Z 453.805,A -85,B 0,C 180,E1 -13780.502,E2 -13780.502} C_VEL
LIN {X 0,Y 347.723,Z 446.003,A -85,B 0,C 180,E1 -13782.251,E2 -13782.251} C_VEL
LIN {X 0,Y 348.494,Z 437.986,A -85,B 0,C 180,E1 -13783.706,E2 -13783.706} C_VEL
LIN {X 0,Y 349.459,Z 428.199,A -85,B 0,C 180,E1 -13785.154,E2 -13785.154} C_VEL
LIN {X 0,Y 350.349,Z 417.321,A -85,B 0,C 180,E1 -13786.458,E2 -13786.458} C_VEL
LIN {X 0,Y 351.385,Z 406.806,A -85,B 0,C 180,E1 -13787.456,E2 -13787.456} C_VEL
LIN {X 0,Y 352.353,Z 394.202,A -85,B 0,C 180,E1 -13788.382,E2 -13788.382} C_VEL
LIN {X 0,Y 353.27,Z 381.072,A -85,B 0,C 180,E1 -13789.085,E2 -13789.085} C_VEL
LIN {X 0,Y 353.824,Z 367.93,A -85,B 0,C 180,E1 -13789.544,E2 -13789.544} C_VEL
LIN {X 0,Y 355.188,Z 297.497,A -85,B 0,C 180,E1 -13791.132,E2 -13791.132} C_VEL
LIN {X 0,Y 350.249,Z 261.768,A -85,B 0,C 180,E1 -13792.251,E2 -13792.251} C_VEL
LIN {X 0,Y 351.791,Z 246.207,A -85,B 0,C 180,E1 -13795.792,E2 -13795.792} C_VEL
LIN {X 0,Y 349.716,Z 234.961,A -85,B 0,C 180,E1 -13798.589,E2 -13798.589} C_VEL
LIN {X 0,Y 347.782,Z 226.164,A -85,B 0,C 180,E1 -13800.887,E2 -13800.887} C_VEL
LIN {X 0,Y 347.733,Z 226.168,A -85,B 0,C 180,E1 -13804.461,E2 -13804.461} C_VEL
LIN {X 0,Y 347.759,Z 226.169,A -85,B 0,C 180,E1 -13807.985,E2 -13807.985} C_VEL
LIN {X 0,Y 347.733,Z 226.172,A -85,B 0,C 180,E1 -13811.827,E2 -13811.827} C_VEL
LIN {X 0,Y 347.684,Z 226.173,A -85,B 0,C 180,E1 -13815.024,E2 -13815.024} C_VEL
LIN {X 0,Y 347.728,Z 226.168,A -85,B 0,C 180,E1 -13818.394,E2 -13818.394} C_VEL
LIN {X 0,Y 347.746,Z 226.167,A -85,B 0,C 180,E1 -13822.009,E2 -13822.009} C_VEL
LIN {X 0,Y 347.717,Z 226.174,A -85,B 0,C 180,E1 -13825.533,E2 -13825.533} C_VEL
LIN {X 0,Y 347.712,Z 226.169,A -85,B 0,C 180,E1 -13828.297,E2 -13828.297} C_VEL
LIN {X 0,Y 347.77,Z 226.162,A -85,B 0,C 180,E1 -13832.302,E2 -13832.302} C_VEL
LIN {X 0,Y 347.783,Z 226.167,A -85,B 0,C 180,E1 -13835.403,E2 -13835.403} C_VEL
LIN {X 0,Y 347.744,Z 226.166,A -85,B 0,C 180,E1 -13838.667,E2 -13838.667} C_VEL
LIN {X 0,Y 347.805,Z 226.158,A -85,B 0,C 180,E1 -13842.356,E2 -13842.356} C_VEL
LIN {X 0,Y 347.862,Z 226.151,A -85,B 0,C 180,E1 -13845.969,E2 -13845.969} C_VEL
LIN {X 0,Y 347.89,Z 226.149,A -85,B 0,C 180,E1 -13849.524,E2 -13849.524} C_VEL
LIN {X 0,Y 348.046,Z 226.134,A -85,B 0,C 180,E1 -13853.041,E2 -13853.041} C_VEL
LIN {X 0,Y 348.16,Z 226.114,A -85,B 0,C 180,E1 -13857.686,E2 -13857.686} C_VEL
LIN {X 0,Y 348.243,Z 226.103,A -85,B 0,C 180,E1 -13860,E2 -13860} C_VEL
LIN {X 0,Y 348.161,Z 226.114,A -85,B 0,C 180,E1 -13862.313,E2 -13862.313} C_VEL
LIN {X 0,Y 348.058,Z 226.131,A -85,B 0,C 180,E1 -13866.958,E2 -13866.958} C_VEL
LIN {X 0,Y 347.89,Z 226.15,A -85,B 0,C 180,E1 -13870.475,E2 -13870.475} C_VEL
LIN {X 0,Y 347.862,Z 226.152,A -85,B 0,C 180,E1 -13874.151,E2 -13874.151} C_VEL
LIN {X 0,Y 347.855,Z 226.154,A -85,B 0,C 180,E1 -13878.292,E2 -13878.292} C_VEL
LIN {X 0,Y 347.805,Z 226.158,A -85,B 0,C 180,E1 -13881.658,E2 -13881.658} C_VEL
LIN {X 0,Y 347.786,Z 226.161,A -85,B 0,C 180,E1 -13885.11,E2 -13885.11} C_VEL
LIN {X 0,Y 347.778,Z 226.161,A -85,B 0,C 180,E1 -13887.696,E2 -13887.696} C_VEL
LIN {X 0,Y 347.732,Z 226.173,A -85,B 0,C 180,E1 -13890.349,E2 -13890.349} C_VEL
LIN {X 0,Y 347.715,Z 226.173,A -85,B 0,C 180,E1 -13894.467,E2 -13894.467} C_VEL
LIN {X 0,Y 347.748,Z 226.169,A -85,B 0,C 180,E1 -13897.991,E2 -13897.991} C_VEL
LIN {X 0,Y 347.761,Z 226.164,A -85,B 0,C 180,E1 -13901.612,E2 -13901.612} C_VEL
LIN {X 0,Y 347.752,Z 226.164,A -85,B 0,C 180,E1 -13905.018,E2 -13905.018} C_VEL
LIN {X 0,Y 347.742,Z 226.168,A -85,B 0,C 180,E1 -13908.398,E2 -13908.398} C_VEL
LIN {X 0,Y 347.757,Z 226.169,A -85,B 0,C 180,E1 -13912.014,E2 -13912.014} C_VEL
LIN {X 0,Y 347.729,Z 226.17,A -85,B 0,C 180,E1 -13915.539,E2 -13915.539} C_VEL
LIN {X 0,Y 347.752,Z 226.169,A -85,B 0,C 180,E1 -13919.656,E2 -13919.656} C_VEL
LIN {X 0,Y 347.842,Z 226.153,A -85,B 0,C 180,E1 -13922.747,E2 -13922.747} C_VEL
LIN {X 0,Y 347.78,Z 226.162,A -85,B 0,C 180,E1 -13926.164,E2 -13926.164} C_VEL
LIN {X 0,Y 347.811,Z 226.16,A -85,B 0,C 180,E1 -13929.912,E2 -13929.912} C_VEL
LIN {X 0,Y 347.861,Z 226.151,A -85,B 0,C 180,E1 -13932.361,E2 -13932.361} C_VEL
LIN {X 0,Y 347.893,Z 226.148,A -85,B 0,C 180,E1 -13935.972,E2 -13935.972} C_VEL
LIN {X 0,Y 347.925,Z 226.147,A -85,B 0,C 180,E1 -13939.527,E2 -13939.527} C_VEL
LIN {X 0,Y 348.089,Z 226.125,A -85,B 0,C 180,E1 -13943.043,E2 -13943.043} C_VEL
LIN {X 0,Y 348.206,Z 226.11,A -85,B 0,C 180,E1 -13947.687,E2 -13947.687} C_VEL
LIN {X 0,Y 348.343,Z 226.091,A -85,B 0,C 180,E1 -13950,E2 -13950} C_VEL
LIN {X 0,Y 348.207,Z 226.108,A -85,B 0,C 180,E1 -13952.313,E2 -13952.313} C_VEL
LIN {X 0,Y 348.083,Z 226.128,A -85,B 0,C 180,E1 -13956.957,E2 -13956.957} C_VEL
LIN {X 0,Y 347.926,Z 226.144,A -85,B 0,C 180,E1 -13960.473,E2 -13960.473} C_VEL
LIN {X 0,Y 347.895,Z 226.147,A -85,B 0,C 180,E1 -13964.149,E2 -13964.149} C_VEL
LIN {X 0,Y 347.885,Z 226.149,A -85,B 0,C 180,E1 -13968.288,E2 -13968.288} C_VEL
LIN {X 0,Y 347.761,Z 226.163,A -85,B 0,C 180,E1 -13971.624,E2 -13971.624} C_VEL
LIN {X 0,Y 347.806,Z 226.163,A -85,B 0,C 180,E1 -13975.106,E2 -13975.106} C_VEL
LIN {X 0,Y 347.891,Z 226.263,A -85,B 0,C 180,E1 -13976.418,E2 -13976.418} C_VEL
LIN {X 0,Y 348.836,Z 231.046,A -85,B 0,C 180,E1 -13977.767,E2 -13977.767} C_VEL
LIN {X 0,Y 354.108,Z 247.007,A -85,B 0,C 180,E1 -13978.443,E2 -13978.443} C_VEL
LIN {X 0,Y 355.88,Z 256.822,A -85,B 0,C 180,E1 -13978.772,E2 -13978.772} C_VEL
LIN {X 0,Y 353.995,Z 338.747,A -85,B 0,C 180,E1 -13980.618,E2 -13980.618} C_VEL
LIN {X 0,Y 353.388,Z 352.346,A -85,B 0,C 180,E1 -13981.154,E2 -13981.154} C_VEL
LIN {X 0,Y 352.839,Z 364.787,A -85,B 0,C 180,E1 -13981.881,E2 -13981.881} C_VEL
LIN {X 0,Y 352.015,Z 376.432,A -85,B 0,C 180,E1 -13982.788,E2 -13982.788} C_VEL
LIN {X 0,Y 351.059,Z 388.057,A -85,B 0,C 180,E1 -13983.95,E2 -13983.95} C_VEL
LIN {X 0,Y 350.232,Z 397.514,A -85,B 0,C 180,E1 -13985.124,E2 -13985.124} C_VEL
LIN {X 0,Y 349.775,Z 402.191,A -85,B 0,C 180,E1 -13985.796,E2 -13985.796} C_VEL
LIN {X 0,Y 348.627,Z 406.494,A -85,B 0,C 180,E1 -13986.436,E2 -13986.436} C_VEL
LIN {X 0,Y 345.145,Z 413.068,A -85,B 0,C 180,E1 -13987.522,E2 -13987.522} C_VEL
LIN {X 0,Y 341.744,Z 419.021,A -85,B 0,C 180,E1 -13988.718,E2 -13988.718} C_VEL
LIN {X 0,Y 340.737,Z 422.35,A -85,B 0,C 180,E1 -13989.522,E2 -13989.522} C_VEL
LIN {X 0,Y 340.096,Z 428.827,A -85,B 0,C 180,E1 -13991.391,E2 -13991.391} C_VEL
LIN {X 0,Y 339.725,Z 433.358,A -85,B 0,C 180,E1 -13993.048,E2 -13993.048} C_VEL
LIN {X 0,Y 339.422,Z 436.977,A -85,B 0,C 180,E1 -13994.742,E2 -13994.742} C_VEL
LIN {X 0,Y 339.089,Z 440.184,A -85,B 0,C 180,E1 -13996.847,E2 -13996.847} C_VEL
LIN {X 0,Y 338.993,Z 441.685,A -85,B 0,C 180,E1 -13998.439,E2 -13998.439} C_VEL
LIN {X 0,Y 338.963,Z 442.479,A -85,B 0,C 180,E1 -14000.091,E2 -14000.091} C_VEL
LIN {X 0,Y 339.016,Z 442.421,A -85,B 0,C 180,E1 -14001.969,E2 -14001.969} C_VEL
LIN {X 0,Y 339.241,Z 441.301,A -85,B 0,C 180,E1 -14003.888,E2 -14003.888} C_VEL
LIN {X 0,Y 339.684,Z 438.751,A -85,B 0,C 180,E1 -14006.04,E2 -14006.04} C_VEL
LIN {X 0,Y 340.225,Z 435.453,A -85,B 0,C 180,E1 -14007.87,E2 -14007.87} C_VEL
LIN {X 0,Y 340.997,Z 430.353,A -85,B 0,C 180,E1 -14009.944,E2 -14009.944} C_VEL
LIN {X 0,Y 341.925,Z 424.359,A -85,B 0,C 180,E1 -14011.788,E2 -14011.788} C_VEL
LIN {X 0,Y 343.215,Z 416.246,A -85,B 0,C 180,E1 -14013.745,E2 -14013.745} C_VEL
LIN {X 0,Y 344.362,Z 408.384,A -85,B 0,C 180,E1 -14015.268,E2 -14015.268} C_VEL
LIN {X 0,Y 345.682,Z 398.205,A -85,B 0,C 180,E1 -14016.858,E2 -14016.858} C_VEL
LIN {X 0,Y 347.055,Z 387.765,A -85,B 0,C 180,E1 -14018.155,E2 -14018.155} C_VEL
LIN {X 0,Y 348.216,Z 377.688,A -85,B 0,C 180,E1 -14019.163,E2 -14019.163} C_VEL
LIN {X 0,Y 349.282,Z 365.908,A -85,B 0,C 180,E1 -14020.099,E2 -14020.099} C_VEL
LIN {X 0,Y 350.225,Z 352.29,A -85,B 0,C 180,E1 -14020.892,E2 -14020.892} C_VEL
LIN {X 0,Y 350.825,Z 339.439,A -85,B 0,C 180,E1 -14021.396,E2 -14021.396} C_VEL
LIN {X 0,Y 353.34,Z 258.911,A -85,B 0,C 180,E1 -14023.312,E2 -14023.312} C_VEL
LIN {X 0,Y 352.111,Z 254.744,A -85,B 0,C 180,E1 -14023.532,E2 -14023.532} C_VEL
LIN {X 0,Y 345.589,Z 239.584,A -85,B 0,C 180,E1 -14024.566,E2 -14024.566} C_VEL
LIN {X 0,Y 342.331,Z 232.842,A -85,B 0,C 180,E1 -14025.104,E2 -14025.104} C_VEL
LIN {X 0,Y 340.823,Z 227.038,A -85,B 0,C 180,E1 -14026.89,E2 -14026.89} C_VEL
LIN {X 0,Y 340.876,Z 227.028,A -85,B 0,C 180,E1 -14030.507,E2 -14030.507} C_VEL
LIN {X 0,Y 341.023,Z 227.008,A -85,B 0,C 180,E1 -14032.898,E2 -14032.898} C_VEL
LIN {X 0,Y 341.124,Z 226.995,A -85,B 0,C 180,E1 -14037.639,E2 -14037.639} C_VEL
LIN {X 0,Y 341.214,Z 226.982,A -85,B 0,C 180,E1 -14040,E2 -14040} C_VEL
LIN {X 0,Y 341.123,Z 226.994,A -85,B 0,C 180,E1 -14042.362,E2 -14042.362} C_VEL
LIN {X 0,Y 341.016,Z 227.009,A -85,B 0,C 180,E1 -14047.103,E2 -14047.103} C_VEL
LIN {X 0,Y 340.834,Z 227.028,A -85,B 0,C 180,E1 -14050.695,E2 -14050.695} C_VEL
LIN {X 0,Y 340.829,Z 227.025,A -85,B 0,C 180,E1 -14054.327,E2 -14054.327} C_VEL
LIN {X 0,Y 340.763,Z 227.037,A -85,B 0,C 180,E1 -14058.448,E2 -14058.448} C_VEL
LIN {X 0,Y 340.687,Z 227.047,A -85,B 0,C 180,E1 -14061.844,E2 -14061.844} C_VEL
LIN {X 0,Y 340.74,Z 227.039,A -85,B 0,C 180,E1 -14065.667,E2 -14065.667} C_VEL
LIN {X 0,Y 340.689,Z 227.048,A -85,B 0,C 180,E1 -14068.325,E2 -14068.325} C_VEL
LIN {X 0,Y 340.664,Z 227.05,A -85,B 0,C 180,E1 -14071.049,E2 -14071.049} C_VEL
LIN {X 0,Y 340.692,Z 227.041,A -85,B 0,C 180,E1 -14075.282,E2 -14075.282} C_VEL
LIN {X 0,Y 340.685,Z 227.045,A -85,B 0,C 180,E1 -14078.389,E2 -14078.389} C_VEL
LIN {X 0,Y 340.677,Z 227.05,A -85,B 0,C 180,E1 -14082.048,E2 -14082.048} C_VEL
LIN {X 0,Y 340.634,Z 227.054,A -85,B 0,C 180,E1 -14086.231,E2 -14086.231} C_VEL
LIN {X 0,Y 340.672,Z 227.047,A -85,B 0,C 180,E1 -14089.757,E2 -14089.757} C_VEL
LIN {X 0,Y 340.692,Z 227.046,A -85,B 0,C 180,E1 -14093.261,E2 -14093.261} C_VEL
LIN {X 0,Y 340.703,Z 227.177,A -85,B 0,C 180,E1 -14096.956,E2 -14096.956} C_VEL
LIN {X 0,Y 343.783,Z 238.903,A -85,B 0,C 180,E1 -14100.326,E2 -14100.326} C_VEL
LIN {X 0,Y 345.906,Z 249.487,A -85,B 0,C 180,E1 -14103.127,E2 -14103.127} C_VEL
LIN {X 0,Y 345.872,Z 253.547,A -85,B 0,C 180,E1 -14104.099,E2 -14104.099} C_VEL
LIN {X 0,Y 345.291,Z 258.561,A -85,B 0,C 180,E1 -14105.241,E2 -14105.241} C_VEL
LIN {X 0,Y 349.782,Z 281.783,A -85,B 0,C 180,E1 -14106.309,E2 -14106.309} C_VEL
LIN {X 0,Y 352.28,Z 299.59,A -85,B 0,C 180,E1 -14106.996,E2 -14106.996} C_VEL
LIN {X 0,Y 350.306,Z 369.294,A -85,B 0,C 180,E1 -14108.679,E2 -14108.679} C_VEL
LIN {X 0,Y 349.301,Z 383.125,A -85,B 0,C 180,E1 -14109.232,E2 -14109.232} C_VEL
LIN {X 0,Y 348.215,Z 395.136,A -85,B 0,C 180,E1 -14109.936,E2 -14109.936} C_VEL
LIN {X 0,Y 346.831,Z 407.673,A -85,B 0,C 180,E1 -14110.931,E2 -14110.931} C_VEL
LIN {X 0,Y 345.35,Z 418.948,A -85,B 0,C 180,E1 -14112.075,E2 -14112.075} C_VEL
LIN {X 0,Y 343.978,Z 429.175,A -85,B 0,C 180,E1 -14113.381,E2 -14113.381} C_VEL
LIN {X 0,Y 342.754,Z 438.43,A -85,B 0,C 180,E1 -14114.847,E2 -14114.847} C_VEL
LIN {X 0,Y 341.52,Z 447.496,A -85,B 0,C 180,E1 -14116.615,E2 -14116.615} C_VEL
LIN {X 0,Y 340.442,Z 454.818,A -85,B 0,C 180,E1 -14118.39,E2 -14118.39} C_VEL
LIN {X 0,Y 339.916,Z 459.785,A -85,B 0,C 180,E1 -14119.879,E2 -14119.879} C_VEL
LIN {X 0,Y 339.438,Z 464.639,A -85,B 0,C 180,E1 -14121.667,E2 -14121.667} C_VEL
LIN {X 0,Y 339.164,Z 468.365,A -85,B 0,C 180,E1 -14123.456,E2 -14123.456} C_VEL
LIN {X 0,Y 339.071,Z 471.059,A -85,B 0,C 180,E1 -14125.245,E2 -14125.245} C_VEL
LIN {X 0,Y 339.088,Z 472.336,A -85,B 0,C 180,E1 -14126.435,E2 -14126.435} C_VEL
LIN {X 0,Y 339.16,Z 473.57,A -85,B 0,C 180,E1 -14128.813,E2 -14128.813} C_VEL
LIN {X 0,Y 339.227,Z 473.586,A -85,B 0,C 180,E1 -14130,E2 -14130} C_VEL
LIN {X 0,Y 339.185,Z 473.181,A -85,B 0,C 180,E1 -14131.187,E2 -14131.187} C_VEL
LIN {X 0,Y 339.098,Z 472.315,A -85,B 0,C 180,E1 -14132.375,E2 -14132.375} C_VEL
LIN {X 0,Y 339.101,Z 471.04,A -85,B 0,C 180,E1 -14133.564,E2 -14133.564} C_VEL
LIN {X 0,Y 339.127,Z 468.056,A -85,B 0,C 180,E1 -14135.479,E2 -14135.479} C_VEL
LIN {X 0,Y 339.268,Z 464.469,A -85,B 0,C 180,E1 -14137.139,E2 -14137.139} C_VEL
LIN {X 0,Y 339.516,Z 459.473,A -85,B 0,C 180,E1 -14138.93,E2 -14138.93} C_VEL
LIN {X 0,Y 339.938,Z 453.151,A -85,B 0,C 180,E1 -14140.722,E2 -14140.722} C_VEL
LIN {X 0,Y 340.746,Z 445.243,A -85,B 0,C 180,E1 -14142.506,E2 -14142.506} C_VEL
LIN {X 0,Y 341.576,Z 437.137,A -85,B 0,C 180,E1 -14143.989,E2 -14143.989} C_VEL
LIN {X 0,Y 342.531,Z 427.236,A -85,B 0,C 180,E1 -14145.468,E2 -14145.468} C_VEL
LIN {X 0,Y 343.496,Z 416.197,A -85,B 0,C 180,E1 -14146.796,E2 -14146.796} C_VEL
LIN {X 0,Y 344.671,Z 403.665,A -85,B 0,C 180,E1 -14147.961,E2 -14147.961} C_VEL
LIN {X 0,Y 345.724,Z 391.449,A -85,B 0,C 180,E1 -14148.825,E2 -14148.825} C_VEL
LIN {X 0,Y 346.554,Z 377.834,A -85,B 0,C 180,E1 -14149.508,E2 -14149.508} C_VEL
LIN {X 0,Y 347.104,Z 364.371,A -85,B 0,C 180,E1 -14149.938,E2 -14149.938} C_VEL
LIN {X 0,Y 348.391,Z 298.47,A -85,B 0,C 180,E1 -14151.447,E2 -14151.447} C_VEL
LIN {X 0,Y 343.322,Z 261.454,A -85,B 0,C 180,E1 -14152.644,E2 -14152.644} C_VEL
LIN {X 0,Y 344.762,Z 247.966,A -85,B 0,C 180,E1 -14155.772,E2 -14155.772} C_VEL
LIN {X 0,Y 344.065,Z 242.914,A -85,B 0,C 180,E1 -14157.029,E2 -14157.029} C_VEL
LIN {X 0,Y 341.686,Z 231.429,A -85,B 0,C 180,E1 -14160.002,E2 -14160.002} C_VEL
LIN {X 0,Y 340.717,Z 227.045,A -85,B 0,C 180,E1 -14161.211,E2 -14161.211} C_VEL
LIN {X 0,Y 340.706,Z 227.042,A -85,B 0,C 180,E1 -14165.276,E2 -14165.276} C_VEL
LIN {X 0,Y 340.695,Z 227.045,A -85,B 0,C 180,E1 -14168.382,E2 -14168.382} C_VEL
LIN {X 0,Y 340.682,Z 227.049,A -85,B 0,C 180,E1 -14172.042,E2 -14172.042} C_VEL
LIN {X 0,Y 340.632,Z 227.053,A -85,B 0,C 180,E1 -14176.224,E2 -14176.224} C_VEL
LIN {X 0,Y 340.665,Z 227.053,A -85,B 0,C 180,E1 -14179.75,E2 -14179.75} C_VEL
LIN {X 0,Y 340.679,Z 227.048,A -85,B 0,C 180,E1 -14183.255,E2 -14183.255} C_VEL
LIN {X 0,Y 340.665,Z 227.048,A -85,B 0,C 180,E1 -14186.15,E2 -14186.15} C_VEL
LIN {X 0,Y 340.696,Z 227.043,A -85,B 0,C 180,E1 -14190.324,E2 -14190.324} C_VEL
LIN {X 0,Y 340.76,Z 227.037,A -85,B 0,C 180,E1 -14193.016,E2 -14193.016} C_VEL
LIN {X 0,Y 340.722,Z 227.044,A -85,B 0,C 180,E1 -14195.635,E2 -14195.635} C_VEL
LIN {X 0,Y 340.681,Z 227.05,A -85,B 0,C 180,E1 -14199.47,E2 -14199.47} C_VEL
LIN {X 0,Y 340.755,Z 227.036,A -85,B 0,C 180,E1 -14201.978,E2 -14201.978} C_VEL
LIN {X 0,Y 340.817,Z 227.03,A -85,B 0,C 180,E1 -14205.715,E2 -14205.715} C_VEL
LIN {X 0,Y 340.833,Z 227.03,A -85,B 0,C 180,E1 -14209.305,E2 -14209.305} C_VEL
LIN {X 0,Y 341.015,Z 227.008,A -85,B 0,C 180,E1 -14212.897,E2 -14212.897} C_VEL
LIN {X 0,Y 341.122,Z 226.991,A -85,B 0,C 180,E1 -14217.638,E2 -14217.638} C_VEL
LIN {X 0,Y 341.195,Z 226.981,A -85,B 0,C 180,E1 -14220,E2 -14220} C_VEL
LIN {X 0,Y 341.123,Z 226.991,A -85,B 0,C 180,E1 -14222.361,E2 -14222.361} C_VEL
LIN {X 0,Y 341.025,Z 227.005,A -85,B 0,C 180,E1 -14227.102,E2 -14227.102} C_VEL
LIN {X 0,Y 340.833,Z 227.032,A -85,B 0,C 180,E1 -14230.695,E2 -14230.695} C_VEL
LIN {X 0,Y 340.827,Z 227.03,A -85,B 0,C 180,E1 -14234.326,E2 -14234.326} C_VEL
LIN {X 0,Y 340.802,Z 227.035,A -85,B 0,C 180,E1 -14238.468,E2 -14238.468} C_VEL
LIN {X 0,Y 340.779,Z 227.034,A -85,B 0,C 180,E1 -14241.883,E2 -14241.883} C_VEL
LIN {X 0,Y 340.743,Z 227.038,A -85,B 0,C 180,E1 -14245.666,E2 -14245.666} C_VEL
LIN {X 0,Y 340.709,Z 227.047,A -85,B 0,C 180,E1 -14248.322,E2 -14248.322} C_VEL
LIN {X 0,Y 340.672,Z 227.047,A -85,B 0,C 180,E1 -14251.047,E2 -14251.047} C_VEL
LIN {X 0,Y 340.689,Z 227.044,A -85,B 0,C 180,E1 -14255.282,E2 -14255.282} C_VEL
LIN {X 0,Y 340.686,Z 227.048,A -85,B 0,C 180,E1 -14258.389,E2 -14258.389} C_VEL
LIN {X 0,Y 340.702,Z 227.043,A -85,B 0,C 180,E1 -14261.307,E2 -14261.307} C_VEL
LIN {X 0,Y 340.684,Z 227.046,A -85,B 0,C 180,E1 -14264.538,E2 -14264.538} C_VEL
LIN {X 0,Y 340.679,Z 227.046,A -85,B 0,C 180,E1 -14268.695,E2 -14268.695} C_VEL
LIN {X 0,Y 340.717,Z 227.045,A -85,B 0,C 180,E1 -14271.776,E2 -14271.776} C_VEL
LIN {X 0,Y 340.708,Z 227.045,A -85,B 0,C 180,E1 -14275.598,E2 -14275.598} C_VEL
LIN {X 0,Y 340.691,Z 227.044,A -85,B 0,C 180,E1 -14278.959,E2 -14278.959} C_VEL
LIN {X 0,Y 340.769,Z 227.034,A -85,B 0,C 180,E1 -14282.477,E2 -14282.477} C_VEL
LIN {X 0,Y 340.763,Z 227.041,A -85,B 0,C 180,E1 -14285.642,E2 -14285.642} C_VEL
LIN {X 0,Y 340.742,Z 227.042,A -85,B 0,C 180,E1 -14289.476,E2 -14289.476} C_VEL
LIN {X 0,Y 340.852,Z 227.026,A -85,B 0,C 180,E1 -14291.986,E2 -14291.986} C_VEL
LIN {X 0,Y 340.865,Z 227.026,A -85,B 0,C 180,E1 -14295.707,E2 -14295.707} C_VEL
LIN {X 0,Y 340.868,Z 227.027,A -85,B 0,C 180,E1 -14299.307,E2 -14299.307} C_VEL
LIN {X 0,Y 341.057,Z 227,A -85,B 0,C 180,E1 -14302.899,E2 -14302.899} C_VEL
LIN {X 0,Y 341.168,Z 226.987,A -85,B 0,C 180,E1 -14307.639,E2 -14307.639} C_VEL
LIN {X 0,Y 341.293,Z 226.969,A -85,B 0,C 180,E1 -14310,E2 -14310} C_VEL
LIN {X 0,Y 341.168,Z 226.985,A -85,B 0,C 180,E1 -14312.361,E2 -14312.361} C_VEL
LIN {X 0,Y 341.052,Z 227.005,A -85,B 0,C 180,E1 -14317.102,E2 -14317.102} C_VEL
LIN {X 0,Y 340.868,Z 227.025,A -85,B 0,C 180,E1 -14320.693,E2 -14320.693} C_VEL
LIN {X 0,Y 340.859,Z 227.024,A -85,B 0,C 180,E1 -14324.323,E2 -14324.323} C_VEL
LIN {X 0,Y 340.831,Z 227.029,A -85,B 0,C 180,E1 -14328.465,E2 -14328.465} C_VEL
LIN {X 0,Y 340.711,Z 227.041,A -85,B 0,C 180,E1 -14331.84,E2 -14331.84} C_VEL
LIN {X 0,Y 340.787,Z 227.036,A -85,B 0,C 180,E1 -14335.66,E2 -14335.66} C_VEL
LIN {X 0,Y 340.823,Z 227.145,A -85,B 0,C 180,E1 -14336.15,E2 -14336.15} C_VEL
LIN {X 0,Y 341.688,Z 231.367,A -85,B 0,C 180,E1 -14337.362,E2 -14337.362} C_VEL
LIN {X 0,Y 347.604,Z 249.322,A -85,B 0,C 180,E1 -14338.146,E2 -14338.146} C_VEL
LIN {X 0,Y 349.093,Z 256.985,A -85,B 0,C 180,E1 -14338.415,E2 -14338.415} C_VEL
LIN {X 0,Y 347.155,Z 339.011,A -85,B 0,C 180,E1 -14340.306,E2 -14340.306} C_VEL
LIN {X 0,Y 346.549,Z 352.742,A -85,B 0,C 180,E1 -14340.86,E2 -14340.86} C_VEL
LIN {X 0,Y 345.935,Z 365.659,A -85,B 0,C 180,E1 -14341.636,E2 -14341.636} C_VEL
LIN {X 0,Y 345.037,Z 378.283,A -85,B 0,C 180,E1 -14342.664,E2 -14342.664} C_VEL
LIN {X 0,Y 344.06,Z 389.38,A -85,B 0,C 180,E1 -14343.819,E2 -14343.819} C_VEL
LIN {X 0,Y 343.119,Z 399.582,A -85,B 0,C 180,E1 -14345.152,E2 -14345.152} C_VEL
LIN {X 0,Y 342.093,Z 409.467,A -85,B 0,C 180,E1 -14346.754,E2 -14346.754} C_VEL
LIN {X 0,Y 341.214,Z 418.102,A -85,B 0,C 180,E1 -14348.493,E2 -14348.493} C_VEL
LIN {X 0,Y 340.737,Z 422.35,A -85,B 0,C 180,E1 -14349.522,E2 -14349.522} C_VEL
LIN {X 0,Y 339.748,Z 425.505,A -85,B 0,C 180,E1 -14350.352,E2 -14350.352} C_VEL
LIN {X 0,Y 336.472,Z 430.153,A -85,B 0,C 180,E1 -14351.732,E2 -14351.732} C_VEL
LIN {X 0,Y 333.294,Z 434.147,A -85,B 0,C 180,E1 -14353.191,E2 -14353.191} C_VEL
LIN {X 0,Y 332.473,Z 436.221,A -85,B 0,C 180,E1 -14354.132,E2 -14354.132} C_VEL
LIN {X 0,Y 332.097,Z 439.429,A -85,B 0,C 180,E1 -14356.009,E2 -14356.009} C_VEL
LIN {X 0,Y 331.934,Z 441.5,A -85,B 0,C 180,E1 -14357.814,E2 -14357.814} C_VEL
LIN {X 0,Y 331.874,Z 442.664,A -85,B 0,C 180,E1 -14359.666,E2 -14359.666} C_VEL
LIN {X 0,Y 331.937,Z 442.75,A -85,B 0,C 180,E1 -14362.121,E2 -14362.121} C_VEL
LIN {X 0,Y 332.149,Z 441.963,A -85,B 0,C 180,E1 -14363.669,E2 -14363.669} C_VEL
LIN {X 0,Y 332.461,Z 440.115,A -85,B 0,C 180,E1 -14365.522,E2 -14365.522} C_VEL
LIN {X 0,Y 333.043,Z 436.921,A -85,B 0,C 180,E1 -14367.565,E2 -14367.565} C_VEL
LIN {X 0,Y 333.817,Z 432.215,A -85,B 0,C 180,E1 -14369.666,E2 -14369.666} C_VEL
LIN {X 0,Y 334.874,Z 425.804,A -85,B 0,C 180,E1 -14371.806,E2 -14371.806} C_VEL
LIN {X 0,Y 336.043,Z 418.819,A -85,B 0,C 180,E1 -14373.615,E2 -14373.615} C_VEL
LIN {X 0,Y 337.395,Z 410.254,A -85,B 0,C 180,E1 -14375.38,E2 -14375.38} C_VEL
LIN {X 0,Y 338.7,Z 400.932,A -85,B 0,C 180,E1 -14376.943,E2 -14376.943} C_VEL
LIN {X 0,Y 340.214,Z 390.307,A -85,B 0,C 180,E1 -14378.355,E2 -14378.355} C_VEL
LIN {X 0,Y 341.586,Z 379.209,A -85,B 0,C 180,E1 -14379.527,E2 -14379.527} C_VEL
LIN {X 0,Y 342.804,Z 366.761,A -85,B 0,C 180,E1 -14380.556,E2 -14380.556} C_VEL
LIN {X 0,Y 343.768,Z 353.868,A -85,B 0,C 180,E1 -14381.333,E2 -14381.333} C_VEL
LIN {X 0,Y 344.444,Z 340.405,A -85,B 0,C 180,E1 -14381.891,E2 -14381.891} C_VEL
LIN {X 0,Y 347.037,Z 259.873,A -85,B 0,C 180,E1 -14383.858,E2 -14383.858} C_VEL
LIN {X 0,Y 341.551,Z 246.341,A -85,B 0,C 180,E1 -14384.778,E2 -14384.778} C_VEL
LIN {X 0,Y 335.222,Z 233.373,A -85,B 0,C 180,E1 -14385.817,E2 -14385.817} C_VEL
LIN {X 0,Y 333.76,Z 227.918,A -85,B 0,C 180,E1 -14387.536,E2 -14387.536} C_VEL
LIN {X 0,Y 333.905,Z 227.895,A -85,B 0,C 180,E1 -14391.549,E2 -14391.549} C_VEL
LIN {X 0,Y 333.978,Z 227.884,A -85,B 0,C 180,E1 -14393.961,E2 -14393.961} C_VEL
LIN {X 0,Y 334.062,Z 227.875,A -85,B 0,C 180,E1 -14397.589,E2 -14397.589} C_VEL
LIN {X 0,Y 334.166,Z 227.861,A -85,B 0,C 180,E1 -14400,E2 -14400} C_VEL
LIN {X 0,Y 334.061,Z 227.874,A -85,B 0,C 180,E1 -14402.412,E2 -14402.412} C_VEL
LIN {X 0,Y 333.97,Z 227.879,A -85,B 0,C 180,E1 -14406.04,E2 -14406.04} C_VEL
LIN {X 0,Y 333.814,Z 227.903,A -85,B 0,C 180,E1 -14409.697,E2 -14409.697} C_VEL
LIN {X 0,Y 333.757,Z 227.908,A -85,B 0,C 180,E1 -14413.393,E2 -14413.393} C_VEL
LIN {X 0,Y 333.693,Z 227.913,A -85,B 0,C 180,E1 -14417.149,E2 -14417.149} C_VEL
LIN {X 0,Y 333.629,Z 227.924,A -85,B 0,C 180,E1 -14419.697,E2 -14419.697} C_VEL
LIN {X 0,Y 333.636,Z 227.918,A -85,B 0,C 180,E1 -14423.593,E2 -14423.593} C_VEL
LIN {X 0,Y 333.699,Z 227.914,A -85,B 0,C 180,E1 -14426.25,E2 -14426.25} C_VEL
LIN {X 0,Y 333.642,Z 227.92,A -85,B 0,C 180,E1 -14428.979,E2 -14428.979} C_VEL
LIN {X 0,Y 333.61,Z 227.927,A -85,B 0,C 180,E1 -14433.212,E2 -14433.212} C_VEL
LIN {X 0,Y 333.651,Z 227.921,A -85,B 0,C 180,E1 -14436.143,E2 -14436.143} C_VEL
LIN {X 0,Y 333.624,Z 227.927,A -85,B 0,C 180,E1 -14439.196,E2 -14439.196} C_VEL
LIN {X 0,Y 333.612,Z 227.926,A -85,B 0,C 180,E1 -14442.503,E2 -14442.503} C_VEL
LIN {X 0,Y 333.578,Z 227.93,A -85,B 0,C 180,E1 -14445.958,E2 -14445.958} C_VEL
LIN {X 0,Y 333.633,Z 227.925,A -85,B 0,C 180,E1 -14449.319,E2 -14449.319} C_VEL
LIN {X 0,Y 333.653,Z 227.923,A -85,B 0,C 180,E1 -14453.171,E2 -14453.171} C_VEL
LIN {X 0,Y 333.655,Z 228.068,A -85,B 0,C 180,E1 -14456.301,E2 -14456.301} C_VEL
LIN {X 0,Y 336.626,Z 239.289,A -85,B 0,C 180,E1 -14459.644,E2 -14459.644} C_VEL
LIN {X 0,Y 338.855,Z 249.706,A -85,B 0,C 180,E1 -14462.521,E2 -14462.521} C_VEL
LIN {X 0,Y 339.257,Z 252.527,A -85,B 0,C 180,E1 -14463.254,E2 -14463.254} C_VEL
LIN {X 0,Y 338.669,Z 258.235,A -85,B 0,C 180,E1 -14464.592,E2 -14464.592} C_VEL
LIN {X 0,Y 343.175,Z 280.643,A -85,B 0,C 180,E1 -14465.673,E2 -14465.673} C_VEL
LIN {X 0,Y 345.8,Z 299.246,A -85,B 0,C 180,E1 -14466.426,E2 -14466.426} C_VEL
LIN {X 0,Y 345.869,Z 305.504,A -85,B 0,C 180,E1 -14466.601,E2 -14466.601} C_VEL
LIN {X 0,Y 343.944,Z 368.513,A -85,B 0,C 180,E1 -14468.147,E2 -14468.147} C_VEL
LIN {X 0,Y 342.914,Z 382.427,A -85,B 0,C 180,E1 -14468.709,E2 -14468.709} C_VEL
LIN {X 0,Y 341.691,Z 394.996,A -85,B 0,C 180,E1 -14469.457,E2 -14469.457} C_VEL
LIN {X 0,Y 340.351,Z 406.651,A -85,B 0,C 180,E1 -14470.396,E2 -14470.396} C_VEL
LIN {X 0,Y 338.829,Z 418.003,A -85,B 0,C 180,E1 -14471.562,E2 -14471.562} C_VEL
LIN {X 0,Y 337.347,Z 428.342,A -85,B 0,C 180,E1 -14472.888,E2 -14472.888} C_VEL
LIN {X 0,Y 335.899,Z 438.522,A -85,B 0,C 180,E1 -14474.53,E2 -14474.53} C_VEL
LIN {X 0,Y 334.607,Z 447.524,A -85,B 0,C 180,E1 -14476.334,E2 -14476.334} C_VEL
LIN {X 0,Y 333.469,Z 454.759,A -85,B 0,C 180,E1 -14478.143,E2 -14478.143} C_VEL
LIN {X 0,Y 332.703,Z 461.404,A -85,B 0,C 180,E1 -14480.272,E2 -14480.272} C_VEL
LIN {X 0,Y 332.258,Z 465.811,A -85,B 0,C 180,E1 -14482.098,E2 -14482.098} C_VEL
LIN {X 0,Y 332.026,Z 469.545,A -85,B 0,C 180,E1 -14484.187,E2 -14484.187} C_VEL
LIN {X 0,Y 332.011,Z 472.056,A -85,B 0,C 180,E1 -14486.359,E2 -14486.359} C_VEL
LIN {X 0,Y 332.062,Z 473.247,A -85,B 0,C 180,E1 -14488.787,E2 -14488.787} C_VEL
LIN {X 0,Y 332.135,Z 473.243,A -85,B 0,C 180,E1 -14490,E2 -14490} C_VEL
LIN {X 0,Y 332.089,Z 472.799,A -85,B 0,C 180,E1 -14491.212,E2 -14491.212} C_VEL
LIN {X 0,Y 332.008,Z 471.909,A -85,B 0,C 180,E1 -14492.426,E2 -14492.426} C_VEL
LIN {X 0,Y 332.027,Z 470.612,A -85,B 0,C 180,E1 -14493.64,E2 -14493.64} C_VEL
LIN {X 0,Y 332.042,Z 468.886,A -85,B 0,C 180,E1 -14494.856,E2 -14494.856} C_VEL
LIN {X 0,Y 332.156,Z 465.381,A -85,B 0,C 180,E1 -14496.682,E2 -14496.682} C_VEL
LIN {X 0,Y 332.354,Z 460.731,A -85,B 0,C 180,E1 -14498.511,E2 -14498.511} C_VEL
LIN {X 0,Y 332.832,Z 453.643,A -85,B 0,C 180,E1 -14500.646,E2 -14500.646} C_VEL
LIN {X 0,Y 333.613,Z 445.958,A -85,B 0,C 180,E1 -14502.469,E2 -14502.469} C_VEL
LIN {X 0,Y 334.428,Z 438.084,A -85,B 0,C 180,E1 -14503.984,E2 -14503.984} C_VEL
LIN {X 0,Y 335.51,Z 427.604,A -85,B 0,C 180,E1 -14505.609,E2 -14505.609} C_VEL
LIN {X 0,Y 336.508,Z 416.437,A -85,B 0,C 180,E1 -14506.999,E2 -14506.999} C_VEL
LIN {X 0,Y 337.561,Z 405.831,A -85,B 0,C 180,E1 -14508.039,E2 -14508.039} C_VEL
LIN {X 0,Y 338.689,Z 393.164,A -85,B 0,C 180,E1 -14508.995,E2 -14508.995} C_VEL
LIN {X 0,Y 339.57,Z 379.837,A -85,B 0,C 180,E1 -14509.729,E2 -14509.729} C_VEL
LIN {X 0,Y 340.215,Z 366.357,A -85,B 0,C 180,E1 -14510.202,E2 -14510.202} C_VEL
LIN {X 0,Y 341.625,Z 299.224,A -85,B 0,C 180,E1 -14511.782,E2 -14511.782} C_VEL
LIN {X 0,Y 336.439,Z 261.076,A -85,B 0,C 180,E1 -14513.062,E2 -14513.062} C_VEL
LIN {X 0,Y 337.789,Z 249.082,A -85,B 0,C 180,E1 -14515.905,E2 -14515.905} C_VEL
LIN {X 0,Y 336.724,Z 242.173,A -85,B 0,C 180,E1 -14517.666,E2 -14517.666} C_VEL
LIN {X 0,Y 334.011,Z 229.519,A -85,B 0,C 180,E1 -14521.048,E2 -14521.048} C_VEL
LIN {X 0,Y 333.7,Z 227.92,A -85,B 0,C 180,E1 -14521.509,E2 -14521.509} C_VEL
LIN {X 0,Y 333.674,Z 227.918,A -85,B 0,C 180,E1 -14524.77,E2 -14524.77} C_VEL
LIN {X 0,Y 333.638,Z 227.925,A -85,B 0,C 180,E1 -14527.648,E2 -14527.648} C_VEL
LIN {X 0,Y 333.631,Z 227.923,A -85,B 0,C 180,E1 -14530.764,E2 -14530.764} C_VEL
LIN {X 0,Y 333.574,Z 227.932,A -85,B 0,C 180,E1 -14534.246,E2 -14534.246} C_VEL
LIN {X 0,Y 333.62,Z 227.929,A -85,B 0,C 180,E1 -14537.615,E2 -14537.615} C_VEL
LIN {X 0,Y 333.629,Z 227.925,A -85,B 0,C 180,E1 -14541.199,E2 -14541.199} C_VEL
LIN {X 0,Y 333.65,Z 227.924,A -85,B 0,C 180,E1 -14543.857,E2 -14543.857} C_VEL
LIN {X 0,Y 333.615,Z 227.93,A -85,B 0,C 180,E1 -14547.411,E2 -14547.411} C_VEL
LIN {X 0,Y 333.649,Z 227.923,A -85,B 0,C 180,E1 -14551.022,E2 -14551.022} C_VEL
LIN {X 0,Y 333.698,Z 227.918,A -85,B 0,C 180,E1 -14553.75,E2 -14553.75} C_VEL
LIN {X 0,Y 333.624,Z 227.927,A -85,B 0,C 180,E1 -14557.717,E2 -14557.717} C_VEL
LIN {X 0,Y 333.704,Z 227.917,A -85,B 0,C 180,E1 -14561.584,E2 -14561.584} C_VEL
LIN {X 0,Y 333.773,Z 227.908,A -85,B 0,C 180,E1 -14565.576,E2 -14565.576} C_VEL
LIN {X 0,Y 333.796,Z 227.908,A -85,B 0,C 180,E1 -14569.076,E2 -14569.076} C_VEL
LIN {X 0,Y 333.964,Z 227.885,A -85,B 0,C 180,E1 -14572.746,E2 -14572.746} C_VEL
LIN {X 0,Y 333.76,Z 227.912,A -85,B 0,C 180,E1 -14575.168,E2 -14575.168} C_VEL
LIN {X 0,Y 334.059,Z 227.871,A -85,B 0,C 180,E1 -14577.588,E2 -14577.588} C_VEL
LIN {X 0,Y 334.148,Z 227.859,A -85,B 0,C 180,E1 -14580,E2 -14580} C_VEL
LIN {X 0,Y 334.061,Z 227.871,A -85,B 0,C 180,E1 -14582.411,E2 -14582.411} C_VEL
LIN {X 0,Y 333.956,Z 227.882,A -85,B 0,C 180,E1 -14586.748,E2 -14586.748} C_VEL
LIN {X 0,Y 333.812,Z 227.901,A -85,B 0,C 180,E1 -14589.696,E2 -14589.696} C_VEL
LIN {X 0,Y 333.756,Z 227.908,A -85,B 0,C 180,E1 -14593.393,E2 -14593.393} C_VEL
LIN {X 0,Y 333.709,Z 227.915,A -85,B 0,C 180,E1 -14597.148,E2 -14597.148} C_VEL
LIN {X 0,Y 333.722,Z 227.912,A -85,B 0,C 180,E1 -14599.691,E2 -14599.691} C_VEL
LIN {X 0,Y 333.692,Z 227.916,A -85,B 0,C 180,E1 -14603.588,E2 -14603.588} C_VEL
LIN {X 0,Y 333.71,Z 227.914,A -85,B 0,C 180,E1 -14607.601,E2 -14607.601} C_VEL
LIN {X 0,Y 333.667,Z 227.925,A -85,B 0,C 180,E1 -14610.365,E2 -14610.365} C_VEL
LIN {X 0,Y 333.656,Z 227.922,A -85,B 0,C 180,E1 -14614.776,E2 -14614.776} C_VEL
LIN {X 0,Y 333.653,Z 227.921,A -85,B 0,C 180,E1 -14618.806,E2 -14618.806} C_VEL
LIN {X 0,Y 333.666,Z 227.921,A -85,B 0,C 180,E1 -14622.513,E2 -14622.513} C_VEL
LIN {X 0,Y 333.605,Z 227.932,A -85,B 0,C 180,E1 -14625.963,E2 -14625.963} C_VEL
LIN {X 0,Y 333.636,Z 227.923,A -85,B 0,C 180,E1 -14629.317,E2 -14629.317} C_VEL
LIN {X 0,Y 333.649,Z 227.921,A -85,B 0,C 180,E1 -14633.171,E2 -14633.171} C_VEL
LIN {X 0,Y 333.623,Z 227.924,A -85,B 0,C 180,E1 -14636.794,E2 -14636.794} C_VEL
LIN {X 0,Y 333.691,Z 227.921,A -85,B 0,C 180,E1 -14639.713,E2 -14639.713} C_VEL
LIN {X 0,Y 333.734,Z 227.911,A -85,B 0,C 180,E1 -14642.404,E2 -14642.404} C_VEL
LIN {X 0,Y 333.718,Z 227.913,A -85,B 0,C 180,E1 -14645.093,E2 -14645.093} C_VEL
LIN {X 0,Y 333.675,Z 227.919,A -85,B 0,C 180,E1 -14649.021,E2 -14649.021} C_VEL
LIN {X 0,Y 333.789,Z 227.909,A -85,B 0,C 180,E1 -14651.591,E2 -14651.591} C_VEL
LIN {X 0,Y 333.804,Z 227.907,A -85,B 0,C 180,E1 -14655.578,E2 -14655.578} C_VEL
LIN {X 0,Y 333.831,Z 227.901,A -85,B 0,C 180,E1 -14659.079,E2 -14659.079} C_VEL
LIN {X 0,Y 334.01,Z 227.877,A -85,B 0,C 180,E1 -14662.748,E2 -14662.748} C_VEL
LIN {X 0,Y 333.807,Z 227.906,A -85,B 0,C 180,E1 -14665.17,E2 -14665.17} C_VEL
LIN {X 0,Y 334.105,Z 227.867,A -85,B 0,C 180,E1 -14667.589,E2 -14667.589} C_VEL
LIN {X 0,Y 334.244,Z 227.847,A -85,B 0,C 180,E1 -14670,E2 -14670} C_VEL
LIN {X 0,Y 334.105,Z 227.865,A -85,B 0,C 180,E1 -14672.411,E2 -14672.411} C_VEL
LIN {X 0,Y 334.009,Z 227.876,A -85,B 0,C 180,E1 -14676.039,E2 -14676.039} C_VEL
LIN {X 0,Y 333.968,Z 227.882,A -85,B 0,C 180,E1 -14678.484,E2 -14678.484} C_VEL
LIN {X 0,Y 333.788,Z 227.904,A -85,B 0,C 180,E1 -14682.153,E2 -14682.153} C_VEL
LIN {X 0,Y 333.773,Z 227.906,A -85,B 0,C 180,E1 -14685.885,E2 -14685.885} C_VEL
LIN {X 0,Y 333.79,Z 227.907,A -85,B 0,C 180,E1 -14688.653,E2 -14688.653} C_VEL
LIN {X 0,Y 333.649,Z 227.922,A -85,B 0,C 180,E1 -14692.279,E2 -14692.279} C_VEL
LIN {X 0,Y 333.772,Z 228.09,A -85,B 0,C 180,E1 -14695.891,E2 -14695.891} C_VEL
LIN {X 0,Y 334.496,Z 231.613,A -85,B 0,C 180,E1 -14696.936,E2 -14696.936} C_VEL
LIN {X 0,Y 340.993,Z 250.999,A -85,B 0,C 180,E1 -14697.815,E2 -14697.815} C_VEL
LIN {X 0,Y 342.373,Z 258.217,A -85,B 0,C 180,E1 -14698.074,E2 -14698.074} C_VEL
LIN {X 0,Y 340.344,Z 339.394,A -85,B 0,C 180,E1 -14699.986,E2 -14699.986} C_VEL
LIN {X 0,Y 339.718,Z 352.874,A -85,B 0,C 180,E1 -14700.54,E2 -14700.54} C_VEL
LIN {X 0,Y 339.097,Z 365.63,A -85,B 0,C 180,E1 -14701.315,E2 -14701.315} C_VEL
LIN {X 0,Y 338.175,Z 377.875,A -85,B 0,C 180,E1 -14702.32,E2 -14702.32} C_VEL
LIN {X 0,Y 337.117,Z 390.122,A -85,B 0,C 180,E1 -14703.617,E2 -14703.617} C_VEL
LIN {X 0,Y 336.07,Z 400.868,A -85,B 0,C 180,E1 -14705.073,E2 -14705.073} C_VEL
LIN {X 0,Y 335.013,Z 410.635,A -85,B 0,C 180,E1 -14706.714,E2 -14706.714} C_VEL
LIN {X 0,Y 334.093,Z 419.214,A -85,B 0,C 180,E1 -14708.524,E2 -14708.524} C_VEL
LIN {X 0,Y 333.428,Z 425.808,A -85,B 0,C 180,E1 -14710.252,E2 -14710.252} C_VEL
LIN {X 0,Y 332.832,Z 432.131,A -85,B 0,C 180,E1 -14712.35,E2 -14712.35} C_VEL
LIN {X 0,Y 332.473,Z 436.221,A -85,B 0,C 180,E1 -14714.132,E2 -14714.132} C_VEL
LIN {X 0,Y 331.649,Z 438.084,A -85,B 0,C 180,E1 -14715.089,E2 -14715.089} C_VEL
LIN {X 0,Y 328.524,Z 440.546,A -85,B 0,C 180,E1 -14716.668,E2 -14716.668} C_VEL
LIN {X 0,Y 325.948,Z 441.94,A -85,B 0,C 180,E1 -14717.97,E2 -14717.97} C_VEL
LIN {X 0,Y 324.859,Z 442.658,A -85,B 0,C 180,E1 -14718.992,E2 -14718.992} C_VEL
LIN {X 0,Y 324.776,Z 442.821,A -85,B 0,C 180,E1 -14719.34,E2 -14719.34} C_VEL
LIN {X 0,Y 324.823,Z 443.261,A -85,B 0,C 180,E1 -14721.153,E2 -14721.153} C_VEL
LIN {X 0,Y 324.963,Z 442.732,A -85,B 0,C 180,E1 -14723.141,E2 -14723.141} C_VEL
LIN {X 0,Y 325.313,Z 441.097,A -85,B 0,C 180,E1 -14725.17,E2 -14725.17} C_VEL
LIN {X 0,Y 325.916,Z 438.02,A -85,B 0,C 180,E1 -14727.378,E2 -14727.378} C_VEL
LIN {X 0,Y 326.67,Z 434.001,A -85,B 0,C 180,E1 -14729.369,E2 -14729.369} C_VEL
LIN {X 0,Y 327.699,Z 428.084,A -85,B 0,C 180,E1 -14731.547,E2 -14731.547} C_VEL
LIN {X 0,Y 328.775,Z 421.866,A -85,B 0,C 180,E1 -14733.327,E2 -14733.327} C_VEL
LIN {X 0,Y 330.126,Z 414.081,A -85,B 0,C 180,E1 -14735.115,E2 -14735.115} C_VEL
LIN {X 0,Y 331.513,Z 405.325,A -85,B 0,C 180,E1 -14736.744,E2 -14736.744} C_VEL
LIN {X 0,Y 332.994,Z 395.53,A -85,B 0,C 180,E1 -14738.208,E2 -14738.208} C_VEL
LIN {X 0,Y 334.58,Z 384.119,A -85,B 0,C 180,E1 -14739.561,E2 -14739.561} C_VEL
LIN {X 0,Y 335.903,Z 372.134,A -85,B 0,C 180,E1 -14740.68,E2 -14740.68} C_VEL
LIN {X 0,Y 337.034,Z 359.863,A -85,B 0,C 180,E1 -14741.537,E2 -14741.537} C_VEL
LIN {X 0,Y 337.837,Z 347.229,A -85,B 0,C 180,E1 -14742.18,E2 -14742.18} C_VEL
LIN {X 0,Y 338.411,Z 334.348,A -85,B 0,C 180,E1 -14742.596,E2 -14742.596} C_VEL
LIN {X 0,Y 340.871,Z 261.582,A -85,B 0,C 180,E1 -14744.409,E2 -14744.409} C_VEL
LIN {X 0,Y 334.956,Z 247.563,A -85,B 0,C 180,E1 -14745.417,E2 -14745.417} C_VEL
LIN {X 0,Y 328.107,Z 233.812,A -85,B 0,C 180,E1 -14746.609,E2 -14746.609} C_VEL
LIN {X 0,Y 326.725,Z 228.796,A -85,B 0,C 180,E1 -14748.288,E2 -14748.288} C_VEL
LIN {X 0,Y 326.92,Z 228.766,A -85,B 0,C 180,E1 -14752.589,E2 -14752.589} C_VEL
LIN {X 0,Y 326.953,Z 228.76,A -85,B 0,C 180,E1 -14753.831,E2 -14753.831} C_VEL
LIN {X 0,Y 327.003,Z 228.755,A -85,B 0,C 180,E1 -14757.537,E2 -14757.537} C_VEL
LIN {X 0,Y 327.119,Z 228.739,A -85,B 0,C 180,E1 -14760,E2 -14760} C_VEL
LIN {X 0,Y 327.002,Z 228.754,A -85,B 0,C 180,E1 -14762.464,E2 -14762.464} C_VEL
LIN {X 0,Y 326.926,Z 228.757,A -85,B 0,C 180,E1 -14766.171,E2 -14766.171} C_VEL
LIN {X 0,Y 326.769,Z 228.781,A -85,B 0,C 180,E1 -14769.908,E2 -14769.908} C_VEL
LIN {X 0,Y 326.722,Z 228.783,A -85,B 0,C 180,E1 -14773.687,E2 -14773.687} C_VEL
LIN {X 0,Y 326.639,Z 228.792,A -85,B 0,C 180,E1 -14777.532,E2 -14777.532} C_VEL
LIN {X 0,Y 326.578,Z 228.805,A -85,B 0,C 180,E1 -14781.46,E2 -14781.46} C_VEL
LIN {X 0,Y 326.643,Z 228.796,A -85,B 0,C 180,E1 -14785.488,E2 -14785.488} C_VEL
LIN {X 0,Y 326.614,Z 228.801,A -85,B 0,C 180,E1 -14788.255,E2 -14788.255} C_VEL
LIN {X 0,Y 326.546,Z 228.808,A -85,B 0,C 180,E1 -14791.101,E2 -14791.101} C_VEL
LIN {X 0,Y 326.581,Z 228.805,A -85,B 0,C 180,E1 -14794.023,E2 -14794.023} C_VEL
LIN {X 0,Y 326.603,Z 228.801,A -85,B 0,C 180,E1 -14797.241,E2 -14797.241} C_VEL
LIN {X 0,Y 326.557,Z 228.805,A -85,B 0,C 180,E1 -14801.134,E2 -14801.134} C_VEL
LIN {X 0,Y 326.508,Z 228.812,A -85,B 0,C 180,E1 -14804.746,E2 -14804.746} C_VEL
LIN {X 0,Y 326.56,Z 228.806,A -85,B 0,C 180,E1 -14808.157,E2 -14808.157} C_VEL
LIN {X 0,Y 326.584,Z 228.803,A -85,B 0,C 180,E1 -14811.391,E2 -14811.391} C_VEL
LIN {X 0,Y 326.627,Z 228.798,A -85,B 0,C 180,E1 -14815.24,E2 -14815.24} C_VEL
LIN {X 0,Y 326.664,Z 229.035,A -85,B 0,C 180,E1 -14815.619,E2 -14815.619} C_VEL
LIN {X 0,Y 329.515,Z 239.734,A -85,B 0,C 180,E1 -14818.945,E2 -14818.945} C_VEL
LIN {X 0,Y 331.786,Z 250.01,A -85,B 0,C 180,E1 -14821.884,E2 -14821.884} C_VEL
LIN {X 0,Y 332.447,Z 255.27,A -85,B 0,C 180,E1 -14823.288,E2 -14823.288} C_VEL
LIN {X 0,Y 332.174,Z 257.854,A -85,B 0,C 180,E1 -14823.901,E2 -14823.901} C_VEL
LIN {X 0,Y 336.841,Z 280.922,A -85,B 0,C 180,E1 -14825.062,E2 -14825.062} C_VEL
LIN {X 0,Y 339.497,Z 299.384,A -85,B 0,C 180,E1 -14825.849,E2 -14825.849} C_VEL
LIN {X 0,Y 339.64,Z 304.911,A -85,B 0,C 180,E1 -14826.02,E2 -14826.02} C_VEL
LIN {X 0,Y 337.562,Z 368.779,A -85,B 0,C 180,E1 -14827.631,E2 -14827.631} C_VEL
LIN {X 0,Y 336.497,Z 382.48,A -85,B 0,C 180,E1 -14828.202,E2 -14828.202} C_VEL
LIN {X 0,Y 335.205,Z 394.912,A -85,B 0,C 180,E1 -14828.961,E2 -14828.961} C_VEL
LIN {X 0,Y 333.711,Z 407.297,A -85,B 0,C 180,E1 -14829.99,E2 -14829.99} C_VEL
LIN {X 0,Y 332.117,Z 418.478,A -85,B 0,C 180,E1 -14831.175,E2 -14831.175} C_VEL
LIN {X 0,Y 330.586,Z 428.62,A -85,B 0,C 180,E1 -14832.527,E2 -14832.527} C_VEL
LIN {X 0,Y 329.124,Z 438.172,A -85,B 0,C 180,E1 -14834.11,E2 -14834.11} C_VEL
LIN {X 0,Y 327.933,Z 446.168,A -85,B 0,C 180,E1 -14835.733,E2 -14835.733} C_VEL
LIN {X 0,Y 326.668,Z 453.615,A -85,B 0,C 180,E1 -14837.577,E2 -14837.577} C_VEL
LIN {X 0,Y 325.87,Z 459.607,A -85,B 0,C 180,E1 -14839.438,E2 -14839.438} C_VEL
LIN {X 0,Y 325.325,Z 464.346,A -85,B 0,C 180,E1 -14841.303,E2 -14841.303} C_VEL
LIN {X 0,Y 325.039,Z 467.976,A -85,B 0,C 180,E1 -14843.171,E2 -14843.171} C_VEL
LIN {X 0,Y 324.889,Z 470.583,A -85,B 0,C 180,E1 -14845.037,E2 -14845.037} C_VEL
LIN {X 0,Y 324.913,Z 471.778,A -85,B 0,C 180,E1 -14846.28,E2 -14846.28} C_VEL
LIN {X 0,Y 324.896,Z 472.549,A -85,B 0,C 180,E1 -14847.521,E2 -14847.521} C_VEL
LIN {X 0,Y 324.965,Z 472.924,A -85,B 0,C 180,E1 -14848.761,E2 -14848.761} C_VEL
LIN {X 0,Y 325.043,Z 472.898,A -85,B 0,C 180,E1 -14850,E2 -14850} C_VEL
LIN {X 0,Y 324.993,Z 472.411,A -85,B 0,C 180,E1 -14851.239,E2 -14851.239} C_VEL
LIN {X 0,Y 324.922,Z 471.501,A -85,B 0,C 180,E1 -14852.479,E2 -14852.479} C_VEL
LIN {X 0,Y 324.954,Z 470.183,A -85,B 0,C 180,E1 -14853.72,E2 -14853.72} C_VEL
LIN {X 0,Y 325.024,Z 466.73,A -85,B 0,C 180,E1 -14855.92,E2 -14855.92} C_VEL
LIN {X 0,Y 325.216,Z 461.836,A -85,B 0,C 180,E1 -14858.074,E2 -14858.074} C_VEL
LIN {X 0,Y 325.657,Z 455.254,A -85,B 0,C 180,E1 -14860.255,E2 -14860.255} C_VEL
LIN {X 0,Y 326.345,Z 448,A -85,B 0,C 180,E1 -14862.119,E2 -14862.119} C_VEL
LIN {X 0,Y 327.28,Z 438.94,A -85,B 0,C 180,E1 -14863.978,E2 -14863.978} C_VEL
LIN {X 0,Y 328.334,Z 429.19,A -85,B 0,C 180,E1 -14865.585,E2 -14865.585} C_VEL
LIN {X 0,Y 329.396,Z 417.955,A -85,B 0,C 180,E1 -14867.058,E2 -14867.058} C_VEL
LIN {X 0,Y 330.603,Z 406.212,A -85,B 0,C 180,E1 -14868.272,E2 -14868.272} C_VEL
LIN {X 0,Y 331.76,Z 393.757,A -85,B 0,C 180,E1 -14869.247,E2 -14869.247} C_VEL
LIN {X 0,Y 332.708,Z 380.047,A -85,B 0,C 180,E1 -14870.033,E2 -14870.033} C_VEL
LIN {X 0,Y 333.39,Z 366.968,A -85,B 0,C 180,E1 -14870.513,E2 -14870.513} C_VEL
LIN {X 0,Y 334.809,Z 299.55,A -85,B 0,C 180,E1 -14872.145,E2 -14872.145} C_VEL
LIN {X 0,Y 329.572,Z 260.794,A -85,B 0,C 180,E1 -14873.469,E2 -14873.469} C_VEL
LIN {X 0,Y 330.797,Z 249.707,A -85,B 0,C 180,E1 -14876.155,E2 -14876.155} C_VEL
LIN {X 0,Y 329.315,Z 241.176,A -85,B 0,C 180,E1 -14878.401,E2 -14878.401} C_VEL
LIN {X 0,Y 326.651,Z 228.798,A -85,B 0,C 180,E1 -14881.807,E2 -14881.807} C_VEL
LIN {X 0,Y 326.6,Z 228.801,A -85,B 0,C 180,E1 -14885.516,E2 -14885.516} C_VEL
LIN {X 0,Y 326.597,Z 228.8,A -85,B 0,C 180,E1 -14889.223,E2 -14889.223} C_VEL
LIN {X 0,Y 326.558,Z 228.804,A -85,B 0,C 180,E1 -14892.968,E2 -14892.968} C_VEL
LIN {X 0,Y 326.556,Z 228.805,A -85,B 0,C 180,E1 -14897.025,E2 -14897.025} C_VEL
LIN {X 0,Y 326.588,Z 228.801,A -85,B 0,C 180,E1 -14900.77,E2 -14900.77} C_VEL
LIN {X 0,Y 326.586,Z 228.801,A -85,B 0,C 180,E1 -14904.477,E2 -14904.477} C_VEL
LIN {X 0,Y 326.579,Z 228.806,A -85,B 0,C 180,E1 -14907.452,E2 -14907.452} C_VEL
LIN {X 0,Y 326.598,Z 228.8,A -85,B 0,C 180,E1 -14910.334,E2 -14910.334} C_VEL
LIN {X 0,Y 326.644,Z 228.796,A -85,B 0,C 180,E1 -14913.138,E2 -14913.138} C_VEL
LIN {X 0,Y 326.615,Z 228.799,A -85,B 0,C 180,E1 -14915.868,E2 -14915.868} C_VEL
LIN {X 0,Y 326.577,Z 228.803,A -85,B 0,C 180,E1 -14919.859,E2 -14919.859} C_VEL
LIN {X 0,Y 326.671,Z 228.792,A -85,B 0,C 180,E1 -14923.758,E2 -14923.758} C_VEL
LIN {X 0,Y 326.72,Z 228.784,A -85,B 0,C 180,E1 -14926.313,E2 -14926.313} C_VEL
LIN {X 0,Y 326.768,Z 228.778,A -85,B 0,C 180,E1 -14930.092,E2 -14930.092} C_VEL
LIN {X 0,Y 326.944,Z 228.757,A -85,B 0,C 180,E1 -14933.829,E2 -14933.829} C_VEL
LIN {X 0,Y 327.001,Z 228.75,A -85,B 0,C 180,E1 -14937.536,E2 -14937.536} C_VEL
LIN {X 0,Y 327.101,Z 228.737,A -85,B 0,C 180,E1 -14940,E2 -14940} C_VEL
LIN {X 0,Y 327.002,Z 228.751,A -85,B 0,C 180,E1 -14942.463,E2 -14942.463} C_VEL
LIN {X 0,Y 326.919,Z 228.758,A -85,B 0,C 180,E1 -14946.741,E2 -14946.741} C_VEL
LIN {X 0,Y 326.768,Z 228.778,A -85,B 0,C 180,E1 -14949.907,E2 -14949.907} C_VEL
LIN {X 0,Y 326.72,Z 228.784,A -85,B 0,C 180,E1 -14953.687,E2 -14953.687} C_VEL
LIN {X 0,Y 326.662,Z 228.791,A -85,B 0,C 180,E1 -14957.529,E2 -14957.529} C_VEL
LIN {X 0,Y 326.654,Z 228.794,A -85,B 0,C 180,E1 -14960.135,E2 -14960.135} C_VEL
LIN {X 0,Y 326.664,Z 228.794,A -85,B 0,C 180,E1 -14962.784,E2 -14962.784} C_VEL
LIN {X 0,Y 326.653,Z 228.794,A -85,B 0,C 180,E1 -14966.86,E2 -14966.86} C_VEL
LIN {X 0,Y 326.609,Z 228.801,A -85,B 0,C 180,E1 -14970.613,E2 -14970.613} C_VEL
LIN {X 0,Y 326.578,Z 228.805,A -85,B 0,C 180,E1 -14974.022,E2 -14974.022} C_VEL
LIN {X 0,Y 326.601,Z 228.799,A -85,B 0,C 180,E1 -14977.241,E2 -14977.241} C_VEL
LIN {X 0,Y 326.611,Z 228.803,A -85,B 0,C 180,E1 -14980.206,E2 -14980.206} C_VEL
LIN {X 0,Y 326.591,Z 228.801,A -85,B 0,C 180,E1 -14983.52,E2 -14983.52} C_VEL
LIN {X 0,Y 326.566,Z 228.803,A -85,B 0,C 180,E1 -14987.029,E2 -14987.029} C_VEL
LIN {X 0,Y 326.598,Z 228.8,A -85,B 0,C 180,E1 -14990.775,E2 -14990.775} C_VEL
LIN {X 0,Y 326.597,Z 228.801,A -85,B 0,C 180,E1 -14994.483,E2 -14994.483} C_VEL
LIN {X 0,Y 326.594,Z 228.802,A -85,B 0,C 180,E1 -14997.458,E2 -14997.458} C_VEL
LIN {X 0,Y 326.649,Z 228.794,A -85,B 0,C 180,E1 -15000.344,E2 -15000.344} C_VEL
LIN {X 0,Y 326.681,Z 228.789,A -85,B 0,C 180,E1 -15004.519,E2 -15004.519} C_VEL
LIN {X 0,Y 326.64,Z 228.794,A -85,B 0,C 180,E1 -15008.547,E2 -15008.547} C_VEL
LIN {X 0,Y 326.739,Z 228.784,A -85,B 0,C 180,E1 -15011.179,E2 -15011.179} C_VEL
LIN {X 0,Y 326.759,Z 228.785,A -85,B 0,C 180,E1 -15015.435,E2 -15015.435} C_VEL
LIN {X 0,Y 326.767,Z 228.779,A -85,B 0,C 180,E1 -15018.84,E2 -15018.84} C_VEL
LIN {X 0,Y 326.964,Z 228.754,A -85,B 0,C 180,E1 -15022.591,E2 -15022.591} C_VEL
LIN {X 0,Y 326.774,Z 228.781,A -85,B 0,C 180,E1 -15025.065,E2 -15025.065} C_VEL
LIN {X 0,Y 327.045,Z 228.747,A -85,B 0,C 180,E1 -15027.537,E2 -15027.537} C_VEL
LIN {X 0,Y 327.196,Z 228.725,A -85,B 0,C 180,E1 -15030,E2 -15030} C_VEL
LIN {X 0,Y 327.046,Z 228.744,A -85,B 0,C 180,E1 -15032.463,E2 -15032.463} C_VEL
LIN {X 0,Y 326.984,Z 228.751,A -85,B 0,C 180,E1 -15036.169,E2 -15036.169} C_VEL
LIN {X 0,Y 326.908,Z 228.763,A -85,B 0,C 180,E1 -15038.654,E2 -15038.654} C_VEL
LIN {X 0,Y 326.731,Z 228.784,A -85,B 0,C 180,E1 -15042.42,E2 -15042.42} C_VEL
LIN {X 0,Y 326.75,Z 228.786,A -85,B 0,C 180,E1 -15044.956,E2 -15044.956} C_VEL
LIN {X 0,Y 326.727,Z 228.789,A -85,B 0,C 180,E1 -15048.836,E2 -15048.836} C_VEL
LIN {X 0,Y 326.596,Z 228.805,A -85,B 0,C 180,E1 -15052.787,E2 -15052.787} C_VEL
LIN {X 0,Y 326.72,Z 228.801,A -85,B 0,C 180,E1 -15055.564,E2 -15055.564} C_VEL
LIN {X 0,Y 327.457,Z 232.202,A -85,B 0,C 180,E1 -15056.528,E2 -15056.528} C_VEL
LIN {X 0,Y 334.532,Z 253.365,A -85,B 0,C 180,E1 -15057.502,E2 -15057.502} C_VEL
LIN {X 0,Y 335.67,Z 259.58,A -85,B 0,C 180,E1 -15057.726,E2 -15057.726} C_VEL
LIN {X 0,Y 333.545,Z 339.465,A -85,B 0,C 180,E1 -15059.65,E2 -15059.65} C_VEL
LIN {X 0,Y 332.903,Z 352.81,A -85,B 0,C 180,E1 -15060.204,E2 -15060.204} C_VEL
LIN {X 0,Y 332.289,Z 364.9,A -85,B 0,C 180,E1 -15060.941,E2 -15060.941} C_VEL
LIN {X 0,Y 331.347,Z 377.373,A -85,B 0,C 180,E1 -15061.961,E2 -15061.961} C_VEL
LIN {X 0,Y 330.274,Z 389.254,A -85,B 0,C 180,E1 -15063.222,E2 -15063.222} C_VEL
LIN {X 0,Y 329.372,Z 398.729,A -85,B 0,C 180,E1 -15064.476,E2 -15064.476} C_VEL
LIN {X 0,Y 328.433,Z 407.411,A -85,B 0,C 180,E1 -15065.869,E2 -15065.869} C_VEL
LIN {X 0,Y 327.423,Z 416.403,A -85,B 0,C 180,E1 -15067.649,E2 -15067.649} C_VEL
LIN {X 0,Y 326.67,Z 422.968,A -85,B 0,C 180,E1 -15069.241,E2 -15069.241} C_VEL
LIN {X 0,Y 326.046,Z 428.963,A -85,B 0,C 180,E1 -15071.025,E2 -15071.025} C_VEL
LIN {X 0,Y 325.615,Z 433.701,A -85,B 0,C 180,E1 -15072.791,E2 -15072.791} C_VEL
LIN {X 0,Y 325.302,Z 437.343,A -85,B 0,C 180,E1 -15074.525,E2 -15074.525} C_VEL
LIN {X 0,Y 324.971,Z 440.017,A -85,B 0,C 180,E1 -15076.208,E2 -15076.208} C_VEL
LIN {X 0,Y 324.833,Z 441.851,A -85,B 0,C 180,E1 -15077.879,E2 -15077.879} C_VEL
LIN {X 0,Y 324.776,Z 442.821,A -85,B 0,C 180,E1 -15079.34,E2 -15079.34} C_VEL
LIN {X 0,Y 324.1,Z 443.215,A -85,B 0,C 180,E1 -15080.376,E2 -15080.376} C_VEL
LIN {X 0,Y 321.209,Z 443.354,A -85,B 0,C 180,E1 -15082.065,E2 -15082.065} C_VEL
LIN {X 0,Y 318.514,Z 442.764,A -85,B 0,C 180,E1 -15083.779,E2 -15083.779} C_VEL
LIN {X 0,Y 318.16,Z 441.975,A -85,B 0,C 180,E1 -15084.835,E2 -15084.835} C_VEL
LIN {X 0,Y 318.663,Z 439.499,A -85,B 0,C 180,E1 -15086.928,E2 -15086.928} C_VEL
LIN {X 0,Y 319.49,Z 435.69,A -85,B 0,C 180,E1 -15089.072,E2 -15089.072} C_VEL
LIN {X 0,Y 320.49,Z 430.228,A -85,B 0,C 180,E1 -15091.29,E2 -15091.29} C_VEL
LIN {X 0,Y 321.572,Z 424.309,A -85,B 0,C 180,E1 -15093.152,E2 -15093.152} C_VEL
LIN {X 0,Y 322.916,Z 417.414,A -85,B 0,C 180,E1 -15094.888,E2 -15094.888} C_VEL
LIN {X 0,Y 324.413,Z 408.453,A -85,B 0,C 180,E1 -15096.712,E2 -15096.712} C_VEL
LIN {X 0,Y 325.914,Z 399.241,A -85,B 0,C 180,E1 -15098.212,E2 -15098.212} C_VEL
LIN {X 0,Y 327.489,Z 388.755,A -85,B 0,C 180,E1 -15099.591,E2 -15099.591} C_VEL
LIN {X 0,Y 328.955,Z 377.788,A -85,B 0,C 180,E1 -15100.742,E2 -15100.742} C_VEL
LIN {X 0,Y 330.211,Z 365.567,A -85,B 0,C 180,E1 -15101.736,E2 -15101.736} C_VEL
LIN {X 0,Y 331.317,Z 352.076,A -85,B 0,C 180,E1 -15102.539,E2 -15102.539} C_VEL
LIN {X 0,Y 332.004,Z 339.155,A -85,B 0,C 180,E1 -15103.043,E2 -15103.043} C_VEL
LIN {X 0,Y 334.691,Z 263.481,A -85,B 0,C 180,E1 -15104.978,E2 -15104.978} C_VEL
LIN {X 0,Y 329.102,Z 250.285,A -85,B 0,C 180,E1 -15105.981,E2 -15105.981} C_VEL
LIN {X 0,Y 322.681,Z 237.621,A -85,B 0,C 180,E1 -15107.133,E2 -15107.133} C_VEL
LIN {X 0,Y 320.918,Z 234.124,A -85,B 0,C 180,E1 -15107.511,E2 -15107.511} C_VEL
LIN {X 0,Y 319.69,Z 229.67,A -85,B 0,C 180,E1 -15109.07,E2 -15109.07} C_VEL
LIN {X 0,Y 319.874,Z 229.643,A -85,B 0,C 180,E1 -15112.425,E2 -15112.425} C_VEL
LIN {X 0,Y 319.706,Z 229.66,A -85,B 0,C 180,E1 -15114.956,E2 -15114.956} C_VEL
LIN {X 0,Y 319.948,Z 229.633,A -85,B 0,C 180,E1 -15117.483,E2 -15117.483} C_VEL
LIN {X 0,Y 320.072,Z 229.617,A -85,B 0,C 180,E1 -15120,E2 -15120} C_VEL
LIN {X 0,Y 319.946,Z 229.633,A -85,B 0,C 180,E1 -15122.518,E2 -15122.518} C_VEL
LIN {X 0,Y 319.885,Z 229.634,A -85,B 0,C 180,E1 -15126.307,E2 -15126.307} C_VEL
LIN {X 0,Y 319.717,Z 229.66,A -85,B 0,C 180,E1 -15130.129,E2 -15130.129} C_VEL
LIN {X 0,Y 319.696,Z 229.657,A -85,B 0,C 180,E1 -15133.994,E2 -15133.994} C_VEL
LIN {X 0,Y 319.587,Z 229.671,A -85,B 0,C 180,E1 -15137.932,E2 -15137.932} C_VEL
LIN {X 0,Y 319.534,Z 229.682,A -85,B 0,C 180,E1 -15141.957,E2 -15141.957} C_VEL
LIN {X 0,Y 319.579,Z 229.674,A -85,B 0,C 180,E1 -15146.093,E2 -15146.093} C_VEL
LIN {X 0,Y 319.536,Z 229.678,A -85,B 0,C 180,E1 -15148.939,E2 -15148.939} C_VEL
LIN {X 0,Y 319.497,Z 229.686,A -85,B 0,C 180,E1 -15151.866,E2 -15151.866} C_VEL
LIN {X 0,Y 319.555,Z 229.674,A -85,B 0,C 180,E1 -15155.545,E2 -15155.545} C_VEL
LIN {X 0,Y 319.54,Z 229.683,A -85,B 0,C 180,E1 -15159.672,E2 -15159.672} C_VEL
LIN {X 0,Y 319.502,Z 229.682,A -85,B 0,C 180,E1 -15163.464,E2 -15163.464} C_VEL
LIN {X 0,Y 319.537,Z 229.681,A -85,B 0,C 180,E1 -15167.02,E2 -15167.02} C_VEL
LIN {X 0,Y 319.533,Z 229.683,A -85,B 0,C 180,E1 -15170.374,E2 -15170.374} C_VEL
LIN {X 0,Y 319.569,Z 229.679,A -85,B 0,C 180,E1 -15174.461,E2 -15174.461} C_VEL
LIN {X 0,Y 319.584,Z 229.741,A -85,B 0,C 180,E1 -15174.797,E2 -15174.797} C_VEL
LIN {X 0,Y 322.664,Z 241.17,A -85,B 0,C 180,E1 -15178.487,E2 -15178.487} C_VEL
LIN {X 0,Y 324.728,Z 250.414,A -85,B 0,C 180,E1 -15181.239,E2 -15181.239} C_VEL
LIN {X 0,Y 325.616,Z 255.166,A -85,B 0,C 180,E1 -15182.577,E2 -15182.577} C_VEL
LIN {X 0,Y 325.662,Z 257.379,A -85,B 0,C 180,E1 -15183.154,E2 -15183.154} C_VEL
LIN {X 0,Y 329.971,Z 278.022,A -85,B 0,C 180,E1 -15184.272,E2 -15184.272} C_VEL
LIN {X 0,Y 333.012,Z 297.535,A -85,B 0,C 180,E1 -15185.161,E2 -15185.161} C_VEL
LIN {X 0,Y 333.509,Z 303.936,A -85,B 0,C 180,E1 -15185.397,E2 -15185.397} C_VEL
LIN {X 0,Y 331.224,Z 368.285,A -85,B 0,C 180,E1 -15187.055,E2 -15187.055} C_VEL
LIN {X 0,Y 330.186,Z 381.924,A -85,B 0,C 180,E1 -15187.64,E2 -15187.64} C_VEL
LIN {X 0,Y 328.876,Z 393.865,A -85,B 0,C 180,E1 -15188.371,E2 -15188.371} C_VEL
LIN {X 0,Y 327.287,Z 406.376,A -85,B 0,C 180,E1 -15189.415,E2 -15189.415} C_VEL
LIN {X 0,Y 325.638,Z 417.658,A -85,B 0,C 180,E1 -15190.622,E2 -15190.622} C_VEL
LIN {X 0,Y 323.98,Z 427.913,A -85,B 0,C 180,E1 -15191.996,E2 -15191.996} C_VEL
LIN {X 0,Y 322.486,Z 437.187,A -85,B 0,C 180,E1 -15193.544,E2 -15193.544} C_VEL
LIN {X 0,Y 321.045,Z 446.271,A -85,B 0,C 180,E1 -15195.421,E2 -15195.421} C_VEL
LIN {X 0,Y 319.735,Z 453.622,A -85,B 0,C 180,E1 -15197.304,E2 -15197.304} C_VEL
LIN {X 0,Y 318.86,Z 459.514,A -85,B 0,C 180,E1 -15199.203,E2 -15199.203} C_VEL
LIN {X 0,Y 318.297,Z 464.187,A -85,B 0,C 180,E1 -15201.11,E2 -15201.11} C_VEL
LIN {X 0,Y 317.973,Z 467.774,A -85,B 0,C 180,E1 -15203.018,E2 -15203.018} C_VEL
LIN {X 0,Y 317.806,Z 470.345,A -85,B 0,C 180,E1 -15204.926,E2 -15204.926} C_VEL
LIN {X 0,Y 317.819,Z 471.501,A -85,B 0,C 180,E1 -15206.197,E2 -15206.197} C_VEL
LIN {X 0,Y 317.813,Z 472.251,A -85,B 0,C 180,E1 -15207.465,E2 -15207.465} C_VEL
LIN {X 0,Y 317.868,Z 472.603,A -85,B 0,C 180,E1 -15208.733,E2 -15208.733} C_VEL
LIN {X 0,Y 317.951,Z 472.539,A -85,B 0,C 180,E1 -15210,E2 -15210} C_VEL
LIN {X 0,Y 317.898,Z 472.014,A -85,B 0,C 180,E1 -15211.267,E2 -15211.267} C_VEL
LIN {X 0,Y 317.839,Z 471.079,A -85,B 0,C 180,E1 -15212.534,E2 -15212.534} C_VEL
LIN {X 0,Y 317.882,Z 469.734,A -85,B 0,C 180,E1 -15213.802,E2 -15213.802} C_VEL
LIN {X 0,Y 317.925,Z 466.563,A -85,B 0,C 180,E1 -15215.863,E2 -15215.863} C_VEL
LIN {X 0,Y 318.059,Z 462.843,A -85,B 0,C 180,E1 -15217.618,E2 -15217.618} C_VEL
LIN {X 0,Y 318.463,Z 456.649,A -85,B 0,C 180,E1 -15219.847,E2 -15219.847} C_VEL
LIN {X 0,Y 319.024,Z 449.829,A -85,B 0,C 180,E1 -15221.756,E2 -15221.756} C_VEL
LIN {X 0,Y 319.944,Z 441.352,A -85,B 0,C 180,E1 -15223.657,E2 -15223.657} C_VEL
LIN {X 0,Y 320.92,Z 432.596,A -85,B 0,C 180,E1 -15225.234,E2 -15225.234} C_VEL
LIN {X 0,Y 322.065,Z 421.802,A -85,B 0,C 180,E1 -15226.804,E2 -15226.804} C_VEL
LIN {X 0,Y 323.174,Z 411.106,A -85,B 0,C 180,E1 -15228.05,E2 -15228.05} C_VEL
LIN {X 0,Y 324.387,Z 399.231,A -85,B 0,C 180,E1 -15229.126,E2 -15229.126} C_VEL
LIN {X 0,Y 325.402,Z 387.008,A -85,B 0,C 180,E1 -15229.967,E2 -15229.967} C_VEL
LIN {X 0,Y 326.243,Z 373.791,A -85,B 0,C 180,E1 -15230.612,E2 -15230.612} C_VEL
LIN {X 0,Y 326.826,Z 358.09,A -85,B 0,C 180,E1 -15231.068,E2 -15231.068} C_VEL
LIN {X 0,Y 328.039,Z 300.307,A -85,B 0,C 180,E1 -15232.493,E2 -15232.493} C_VEL
LIN {X 0,Y 322.712,Z 260.467,A -85,B 0,C 180,E1 -15233.899,E2 -15233.899} C_VEL
LIN {X 0,Y 323.775,Z 251.683,A -85,B 0,C 180,E1 -15236.072,E2 -15236.072} C_VEL
LIN {X 0,Y 323.322,Z 247.554,A -85,B 0,C 180,E1 -15237.156,E2 -15237.156} C_VEL
LIN {X 0,Y 321.046,Z 236.363,A -85,B 0,C 180,E1 -15240.227,E2 -15240.227} C_VEL
LIN {X 0,Y 319.584,Z 229.678,A -85,B 0,C 180,E1 -15242.13,E2 -15242.13} C_VEL
LIN {X 0,Y 319.546,Z 229.68,A -85,B 0,C 180,E1 -15246.424,E2 -15246.424} C_VEL
LIN {X 0,Y 319.546,Z 229.681,A -85,B 0,C 180,E1 -15249.665,E2 -15249.665} C_VEL
LIN {X 0,Y 319.504,Z 229.686,A -85,B 0,C 180,E1 -15253.457,E2 -15253.457} C_VEL
LIN {X 0,Y 319.534,Z 229.68,A -85,B 0,C 180,E1 -15257.013,E2 -15257.013} C_VEL
LIN {X 0,Y 319.525,Z 229.681,A -85,B 0,C 180,E1 -15260.367,E2 -15260.367} C_VEL
LIN {X 0,Y 319.533,Z 229.685,A -85,B 0,C 180,E1 -15263.568,E2 -15263.568} C_VEL
LIN {X 0,Y 319.552,Z 229.677,A -85,B 0,C 180,E1 -15266.683,E2 -15266.683} C_VEL
LIN {X 0,Y 319.535,Z 229.684,A -85,B 0,C 180,E1 -15269.61,E2 -15269.61} C_VEL
LIN {X 0,Y 319.569,Z 229.675,A -85,B 0,C 180,E1 -15272.494,E2 -15272.494} C_VEL
LIN {X 0,Y 319.571,Z 229.679,A -85,B 0,C 180,E1 -15275.301,E2 -15275.301} C_VEL
LIN {X 0,Y 319.533,Z 229.68,A -85,B 0,C 180,E1 -15278.043,E2 -15278.043} C_VEL
LIN {X 0,Y 319.578,Z 229.674,A -85,B 0,C 180,E1 -15282.068,E2 -15282.068} C_VEL
LIN {X 0,Y 319.695,Z 229.659,A -85,B 0,C 180,E1 -15286.006,E2 -15286.006} C_VEL
LIN {X 0,Y 319.715,Z 229.657,A -85,B 0,C 180,E1 -15289.871,E2 -15289.871} C_VEL
LIN {X 0,Y 319.899,Z 229.634,A -85,B 0,C 180,E1 -15293.693,E2 -15293.693} C_VEL
LIN {X 0,Y 319.945,Z 229.629,A -85,B 0,C 180,E1 -15297.482,E2 -15297.482} C_VEL
LIN {X 0,Y 320.056,Z 229.613,A -85,B 0,C 180,E1 -15300,E2 -15300} C_VEL
LIN {X 0,Y 319.947,Z 229.63,A -85,B 0,C 180,E1 -15302.517,E2 -15302.517} C_VEL
LIN {X 0,Y 319.879,Z 229.635,A -85,B 0,C 180,E1 -15306.731,E2 -15306.731} C_VEL
LIN {X 0,Y 319.715,Z 229.658,A -85,B 0,C 180,E1 -15310.128,E2 -15310.128} C_VEL
LIN {X 0,Y 319.695,Z 229.663,A -85,B 0,C 180,E1 -15314.724,E2 -15314.724} C_VEL
LIN {X 0,Y 319.647,Z 229.664,A -85,B 0,C 180,E1 -15319.256,E2 -15319.256} C_VEL
LIN {X 0,Y 319.609,Z 229.67,A -85,B 0,C 180,E1 -15323.316,E2 -15323.316} C_VEL
LIN {X 0,Y 319.605,Z 229.673,A -85,B 0,C 180,E1 -15326.09,E2 -15326.09} C_VEL
LIN {X 0,Y 319.558,Z 229.677,A -85,B 0,C 180,E1 -15328.936,E2 -15328.936} C_VEL
LIN {X 0,Y 319.502,Z 229.685,A -85,B 0,C 180,E1 -15331.865,E2 -15331.865} C_VEL
LIN {X 0,Y 319.551,Z 229.677,A -85,B 0,C 180,E1 -15335.545,E2 -15335.545} C_VEL
LIN {X 0,Y 319.557,Z 229.679,A -85,B 0,C 180,E1 -15338.01,E2 -15338.01} C_VEL
LIN {X 0,Y 319.573,Z 229.675,A -85,B 0,C 180,E1 -15341.614,E2 -15341.614} C_VEL
LIN {X 0,Y 319.507,Z 229.683,A -85,B 0,C 180,E1 -15345.267,E2 -15345.267} C_VEL
LIN {X 0,Y 319.515,Z 229.682,A -85,B 0,C 180,E1 -15348.715,E2 -15348.715} C_VEL
LIN {X 0,Y 319.561,Z 229.678,A -85,B 0,C 180,E1 -15352.347,E2 -15352.347} C_VEL
LIN {X 0,Y 319.545,Z 229.678,A -85,B 0,C 180,E1 -15355.126,E2 -15355.126} C_VEL
LIN {X 0,Y 319.558,Z 229.676,A -85,B 0,C 180,E1 -15359.061,E2 -15359.061} C_VEL
LIN {X 0,Y 319.599,Z 229.672,A -85,B 0,C 180,E1 -15362.501,E2 -15362.501} C_VEL
LIN {X 0,Y 319.598,Z 229.674,A -85,B 0,C 180,E1 -15365.307,E2 -15365.307} C_VEL
LIN {X 0,Y 319.59,Z 229.674,A -85,B 0,C 180,E1 -15368.05,E2 -15368.05} C_VEL
LIN {X 0,Y 319.683,Z 229.661,A -85,B 0,C 180,E1 -15370.964,E2 -15370.964} C_VEL
LIN {X 0,Y 319.727,Z 229.659,A -85,B 0,C 180,E1 -15375.277,E2 -15375.277} C_VEL
LIN {X 0,Y 319.754,Z 229.653,A -85,B 0,C 180,E1 -15379.874,E2 -15379.874} C_VEL
LIN {X 0,Y 319.923,Z 229.631,A -85,B 0,C 180,E1 -15382.427,E2 -15382.427} C_VEL
LIN {X 0,Y 319.743,Z 229.656,A -85,B 0,C 180,E1 -15384.957,E2 -15384.957} C_VEL
LIN {X 0,Y 319.989,Z 229.626,A -85,B 0,C 180,E1 -15387.483,E2 -15387.483} C_VEL
LIN {X 0,Y 320.148,Z 229.603,A -85,B 0,C 180,E1 -15390,E2 -15390} C_VEL
LIN {X 0,Y 319.99,Z 229.623,A -85,B 0,C 180,E1 -15392.517,E2 -15392.517} C_VEL
LIN {X 0,Y 319.939,Z 229.629,A -85,B 0,C 180,E1 -15396.305,E2 -15396.305} C_VEL
LIN {X 0,Y 319.836,Z 229.646,A -85,B 0,C 180,E1 -15398.847,E2 -15398.847} C_VEL
LIN {X 0,Y 319.679,Z 229.665,A -85,B 0,C 180,E1 -15402.699,E2 -15402.699} C_VEL
LIN {X 0,Y 319.695,Z 229.662,A -85,B 0,C 180,E1 -15405.294,E2 -15405.294} C_VEL
LIN {X 0,Y 319.646,Z 229.667,A -85,B 0,C 180,E1 -15409.255,E2 -15409.255} C_VEL
LIN {X 0,Y 319.556,Z 229.678,A -85,B 0,C 180,E1 -15413.318,E2 -15413.318} C_VEL
LIN {X 0,Y 319.659,Z 229.821,A -85,B 0,C 180,E1 -15415.312,E2 -15415.312} C_VEL
LIN {X 0,Y 320.23,Z 232.467,A -85,B 0,C 180,E1 -15416.076,E2 -15416.076} C_VEL
LIN {X 0,Y 328.052,Z 255.602,A -85,B 0,C 180,E1 -15417.183,E2 -15417.183} C_VEL
LIN {X 0,Y 328.916,Z 259.935,A -85,B 0,C 180,E1 -15417.348,E2 -15417.348} C_VEL
LIN {X 0,Y 326.686,Z 340.611,A -85,B 0,C 180,E1 -15419.345,E2 -15419.345} C_VEL
LIN {X 0,Y 326.003,Z 354.208,A -85,B 0,C 180,E1 -15419.938,E2 -15419.938} C_VEL
LIN {X 0,Y 325.369,Z 366.167,A -85,B 0,C 180,E1 -15420.702,E2 -15420.702} C_VEL
LIN {X 0,Y 324.466,Z 377.372,A -85,B 0,C 180,E1 -15421.644,E2 -15421.644} C_VEL
LIN {X 0,Y 323.407,Z 389.073,A -85,B 0,C 180,E1 -15422.903,E2 -15422.903} C_VEL
LIN {X 0,Y 322.387,Z 399.279,A -85,B 0,C 180,E1 -15424.275,E2 -15424.275} C_VEL
LIN {X 0,Y 321.437,Z 407.79,A -85,B 0,C 180,E1 -15425.674,E2 -15425.674} C_VEL
LIN {X 0,Y 320.452,Z 416.402,A -85,B 0,C 180,E1 -15427.408,E2 -15427.408} C_VEL
LIN {X 0,Y 319.596,Z 423.662,A -85,B 0,C 180,E1 -15429.209,E2 -15429.209} C_VEL
LIN {X 0,Y 318.975,Z 429.353,A -85,B 0,C 180,E1 -15430.951,E2 -15430.951} C_VEL
LIN {X 0,Y 318.453,Z 435.028,A -85,B 0,C 180,E1 -15433.162,E2 -15433.162} C_VEL
LIN {X 0,Y 318.109,Z 438.563,A -85,B 0,C 180,E1 -15435.011,E2 -15435.011} C_VEL
LIN {X 0,Y 317.804,Z 441.119,A -85,B 0,C 180,E1 -15436.86,E2 -15436.86} C_VEL
LIN {X 0,Y 317.711,Z 442.796,A -85,B 0,C 180,E1 -15438.766,E2 -15438.766} C_VEL
LIN {X 0,Y 317.699,Z 443.553,A -85,B 0,C 180,E1 -15440.73,E2 -15440.73} C_VEL
LIN {X 0,Y 317.827,Z 443.314,A -85,B 0,C 180,E1 -15442.747,E2 -15442.747} C_VEL
LIN {X 0,Y 318.16,Z 441.975,A -85,B 0,C 180,E1 -15444.835,E2 -15444.835} C_VEL
LIN {X 0,Y 317.867,Z 440.97,A -85,B 0,C 180,E1 -15445.88,E2 -15445.88} C_VEL
LIN {X 0,Y 315.524,Z 438.879,A -85,B 0,C 180,E1 -15447.58,E2 -15447.58} C_VEL
LIN {X 0,Y 313.522,Z 436.759,A -85,B 0,C 180,E1 -15448.934,E2 -15448.934} C_VEL
LIN {X 0,Y 312.857,Z 434.794,A -85,B 0,C 180,E1 -15449.954,E2 -15449.954} C_VEL
LIN {X 0,Y 312.916,Z 434.042,A -85,B 0,C 180,E1 -15450.292,E2 -15450.292} C_VEL
LIN {X 0,Y 314.011,Z 428.656,A -85,B 0,C 180,E1 -15452.318,E2 -15452.318} C_VEL
LIN {X 0,Y 315.299,Z 422.145,A -85,B 0,C 180,E1 -15454.237,E2 -15454.237} C_VEL
LIN {X 0,Y 316.978,Z 413.481,A -85,B 0,C 180,E1 -15456.268,E2 -15456.268} C_VEL
LIN {X 0,Y 318.646,Z 403.759,A -85,B 0,C 180,E1 -15458.066,E2 -15458.066} C_VEL
LIN {X 0,Y 320.506,Z 392.793,A -85,B 0,C 180,E1 -15459.669,E2 -15459.669} C_VEL
LIN {X 0,Y 322.072,Z 382.162,A -85,B 0,C 180,E1 -15460.894,E2 -15460.894} C_VEL
LIN {X 0,Y 323.453,Z 370.437,A -85,B 0,C 180,E1 -15461.964,E2 -15461.964} C_VEL
LIN {X 0,Y 324.646,Z 358.188,A -85,B 0,C 180,E1 -15462.809,E2 -15462.809} C_VEL
LIN {X 0,Y 325.464,Z 345.5,A -85,B 0,C 180,E1 -15463.429,E2 -15463.429} C_VEL
LIN {X 0,Y 326.243,Z 325.853,A -85,B 0,C 180,E1 -15464.003,E2 -15464.003} C_VEL
LIN {X 0,Y 328.642,Z 265.482,A -85,B 0,C 180,E1 -15465.566,E2 -15465.566} C_VEL
LIN {X 0,Y 322.964,Z 252.285,A -85,B 0,C 180,E1 -15466.627,E2 -15466.627} C_VEL
LIN {X 0,Y 316.671,Z 240.096,A -85,B 0,C 180,E1 -15467.809,E2 -15467.809} C_VEL
LIN {X 0,Y 313.813,Z 234.762,A -85,B 0,C 180,E1 -15468.372,E2 -15468.372} C_VEL
LIN {X 0,Y 312.699,Z 230.54,A -85,B 0,C 180,E1 -15469.888,E2 -15469.888} C_VEL
LIN {X 0,Y 312.864,Z 230.514,A -85,B 0,C 180,E1 -15473.552,E2 -15473.552} C_VEL
LIN {X 0,Y 312.895,Z 230.511,A -85,B 0,C 180,E1 -15477.426,E2 -15477.426} C_VEL
LIN {X 0,Y 313.028,Z 230.494,A -85,B 0,C 180,E1 -15480,E2 -15480} C_VEL
LIN {X 0,Y 312.892,Z 230.511,A -85,B 0,C 180,E1 -15482.575,E2 -15482.575} C_VEL
LIN {X 0,Y 312.845,Z 230.512,A -85,B 0,C 180,E1 -15486.45,E2 -15486.45} C_VEL
LIN {X 0,Y 312.724,Z 230.528,A -85,B 0,C 180,E1 -15489.052,E2 -15489.052} C_VEL
LIN {X 0,Y 312.598,Z 230.546,A -85,B 0,C 180,E1 -15492.993,E2 -15492.993} C_VEL
LIN {X 0,Y 312.59,Z 230.547,A -85,B 0,C 180,E1 -15495.653,E2 -15495.653} C_VEL
LIN {X 0,Y 312.505,Z 230.556,A -85,B 0,C 180,E1 -15499.715,E2 -15499.715} C_VEL
LIN {X 0,Y 312.507,Z 230.55,A -85,B 0,C 180,E1 -15503.879,E2 -15503.879} C_VEL
LIN {X 0,Y 312.507,Z 230.552,A -85,B 0,C 180,E1 -15506.73,E2 -15506.73} C_VEL
LIN {X 0,Y 312.479,Z 230.554,A -85,B 0,C 180,E1 -15509.657,E2 -15509.657} C_VEL
LIN {X 0,Y 312.496,Z 230.558,A -85,B 0,C 180,E1 -15513.692,E2 -15513.692} C_VEL
LIN {X 0,Y 312.496,Z 230.558,A -85,B 0,C 180,E1 -15517.39,E2 -15517.39} C_VEL
LIN {X 0,Y 312.47,Z 230.559,A -85,B 0,C 180,E1 -15520.713,E2 -15520.713} C_VEL
LIN {X 0,Y 312.433,Z 230.568,A -85,B 0,C 180,E1 -15524.213,E2 -15524.213} C_VEL
LIN {X 0,Y 312.453,Z 230.561,A -85,B 0,C 180,E1 -15527.926,E2 -15527.926} C_VEL
LIN {X 0,Y 312.485,Z 230.561,A -85,B 0,C 180,E1 -15530.974,E2 -15530.974} C_VEL
LIN {X 0,Y 312.535,Z 230.685,A -85,B 0,C 180,E1 -15533.979,E2 -15533.979} C_VEL
LIN {X 0,Y 315.195,Z 240.344,A -85,B 0,C 180,E1 -15537.272,E2 -15537.272} C_VEL
LIN {X 0,Y 317.677,Z 250.71,A -85,B 0,C 180,E1 -15540.509,E2 -15540.509} C_VEL
LIN {X 0,Y 318.959,Z 257.25,A -85,B 0,C 180,E1 -15542.352,E2 -15542.352} C_VEL
LIN {X 0,Y 320.845,Z 264.083,A -85,B 0,C 180,E1 -15542.806,E2 -15542.806} C_VEL
LIN {X 0,Y 324.728,Z 283.883,A -85,B 0,C 180,E1 -15543.874,E2 -15543.874} C_VEL
LIN {X 0,Y 327.155,Z 300.996,A -85,B 0,C 180,E1 -15544.665,E2 -15544.665} C_VEL
LIN {X 0,Y 327.307,Z 305.926,A -85,B 0,C 180,E1 -15544.827,E2 -15544.827} C_VEL
LIN {X 0,Y 324.972,Z 368.028,A -85,B 0,C 180,E1 -15546.461,E2 -15546.461} C_VEL
LIN {X 0,Y 323.834,Z 382.334,A -85,B 0,C 180,E1 -15547.092,E2 -15547.092} C_VEL
LIN {X 0,Y 322.341,Z 395.008,A -85,B 0,C 180,E1 -15547.91,E2 -15547.91} C_VEL
LIN {X 0,Y 320.698,Z 407.184,A -85,B 0,C 180,E1 -15548.973,E2 -15548.973} C_VEL
LIN {X 0,Y 318.982,Z 418.211,A -85,B 0,C 180,E1 -15550.201,E2 -15550.201} C_VEL
LIN {X 0,Y 317.241,Z 428.222,A -85,B 0,C 180,E1 -15551.6,E2 -15551.6} C_VEL
LIN {X 0,Y 315.635,Z 437.627,A -85,B 0,C 180,E1 -15553.227,E2 -15553.227} C_VEL
LIN {X 0,Y 314.166,Z 446.378,A -85,B 0,C 180,E1 -15555.094,E2 -15555.094} C_VEL
LIN {X 0,Y 312.814,Z 453.628,A -85,B 0,C 180,E1 -15557.018,E2 -15557.018} C_VEL
LIN {X 0,Y 311.861,Z 459.447,A -85,B 0,C 180,E1 -15558.958,E2 -15558.958} C_VEL
LIN {X 0,Y 311.243,Z 464.057,A -85,B 0,C 180,E1 -15560.906,E2 -15560.906} C_VEL
LIN {X 0,Y 310.903,Z 467.579,A -85,B 0,C 180,E1 -15562.859,E2 -15562.859} C_VEL
LIN {X 0,Y 310.71,Z 470.098,A -85,B 0,C 180,E1 -15564.809,E2 -15564.809} C_VEL
LIN {X 0,Y 310.728,Z 471.226,A -85,B 0,C 180,E1 -15566.11,E2 -15566.11} C_VEL
LIN {X 0,Y 310.732,Z 471.954,A -85,B 0,C 180,E1 -15567.408,E2 -15567.408} C_VEL
LIN {X 0,Y 310.775,Z 472.282,A -85,B 0,C 180,E1 -15568.704,E2 -15568.704} C_VEL
LIN {X 0,Y 310.86,Z 472.169,A -85,B 0,C 180,E1 -15570,E2 -15570} C_VEL
LIN {X 0,Y 310.804,Z 471.617,A -85,B 0,C 180,E1 -15571.295,E2 -15571.295} C_VEL
LIN {X 0,Y 310.759,Z 470.657,A -85,B 0,C 180,E1 -15572.592,E2 -15572.592} C_VEL
LIN {X 0,Y 310.789,Z 469.281,A -85,B 0,C 180,E1 -15573.889,E2 -15573.889} C_VEL
LIN {X 0,Y 310.836,Z 466.357,A -85,B 0,C 180,E1 -15575.819,E2 -15575.819} C_VEL
LIN {X 0,Y 310.999,Z 462.27,A -85,B 0,C 180,E1 -15577.792,E2 -15577.792} C_VEL
LIN {X 0,Y 311.417,Z 455.974,A -85,B 0,C 180,E1 -15580.072,E2 -15580.072} C_VEL
LIN {X 0,Y 312.037,Z 449.074,A -85,B 0,C 180,E1 -15582.023,E2 -15582.023} C_VEL
LIN {X 0,Y 312.842,Z 442.03,A -85,B 0,C 180,E1 -15583.642,E2 -15583.642} C_VEL
LIN {X 0,Y 313.828,Z 433.529,A -85,B 0,C 180,E1 -15585.254,E2 -15585.254} C_VEL
LIN {X 0,Y 314.977,Z 423.031,A -85,B 0,C 180,E1 -15586.86,E2 -15586.86} C_VEL
LIN {X 0,Y 316.099,Z 412.657,A -85,B 0,C 180,E1 -15588.134,E2 -15588.134} C_VEL
LIN {X 0,Y 317.279,Z 401.371,A -85,B 0,C 180,E1 -15589.236,E2 -15589.236} C_VEL
LIN {X 0,Y 318.395,Z 388.725,A -85,B 0,C 180,E1 -15590.173,E2 -15590.173} C_VEL
LIN {X 0,Y 319.309,Z 375.484,A -85,B 0,C 180,E1 -15590.87,E2 -15590.87} C_VEL
LIN {X 0,Y 319.883,Z 362.906,A -85,B 0,C 180,E1 -15591.294,E2 -15591.294} C_VEL
LIN {X 0,Y 321.304,Z 301.322,A -85,B 0,C 180,E1 -15592.845,E2 -15592.845} C_VEL
LIN {X 0,Y 315.837,Z 260.32,A -85,B 0,C 180,E1 -15594.298,E2 -15594.298} C_VEL
LIN {X 0,Y 316.826,Z 252.262,A -85,B 0,C 180,E1 -15596.334,E2 -15596.334} C_VEL
LIN {X 0,Y 315.411,Z 243.929,A -85,B 0,C 180,E1 -15598.621,E2 -15598.621} C_VEL
LIN {X 0,Y 312.54,Z 230.555,A -85,B 0,C 180,E1 -15602.497,E2 -15602.497} C_VEL
LIN {X 0,Y 312.523,Z 230.558,A -85,B 0,C 180,E1 -15605.946,E2 -15605.946} C_VEL
LIN {X 0,Y 312.49,Z 230.56,A -85,B 0,C 180,E1 -15610.122,E2 -15610.122} C_VEL
LIN {X 0,Y 312.441,Z 230.568,A -85,B 0,C 180,E1 -15613.961,E2 -15613.961} C_VEL
LIN {X 0,Y 312.464,Z 230.564,A -85,B 0,C 180,E1 -15617.916,E2 -15617.916} C_VEL
LIN {X 0,Y 312.48,Z 230.559,A -85,B 0,C 180,E1 -15620.968,E2 -15620.968} C_VEL
LIN {X 0,Y 312.506,Z 230.556,A -85,B 0,C 180,E1 -15624.216,E2 -15624.216} C_VEL
LIN {X 0,Y 312.475,Z 230.562,A -85,B 0,C 180,E1 -15627.33,E2 -15627.33} C_VEL
LIN {X 0,Y 312.536,Z 230.553,A -85,B 0,C 180,E1 -15631.821,E2 -15631.821} C_VEL
LIN {X 0,Y 312.544,Z 230.55,A -85,B 0,C 180,E1 -15634.707,E2 -15634.707} C_VEL
LIN {X 0,Y 312.487,Z 230.559,A -85,B 0,C 180,E1 -15638.909,E2 -15638.909} C_VEL
LIN {X 0,Y 312.532,Z 230.553,A -85,B 0,C 180,E1 -15641.649,E2 -15641.649} C_VEL
LIN {X 0,Y 312.649,Z 230.538,A -85,B 0,C 180,E1 -15645.684,E2 -15645.684} C_VEL
LIN {X 0,Y 312.662,Z 230.537,A -85,B 0,C 180,E1 -15649.64,E2 -15649.64} C_VEL
LIN {X 0,Y 312.806,Z 230.518,A -85,B 0,C 180,E1 -15652.252,E2 -15652.252} C_VEL
LIN {X 0,Y 312.857,Z 230.512,A -85,B 0,C 180,E1 -15653.55,E2 -15653.55} C_VEL
LIN {X 0,Y 312.891,Z 230.507,A -85,B 0,C 180,E1 -15657.425,E2 -15657.425} C_VEL
LIN {X 0,Y 313.013,Z 230.489,A -85,B 0,C 180,E1 -15660,E2 -15660} C_VEL
LIN {X 0,Y 312.893,Z 230.508,A -85,B 0,C 180,E1 -15662.574,E2 -15662.574} C_VEL
LIN {X 0,Y 312.84,Z 230.513,A -85,B 0,C 180,E1 -15666.713,E2 -15666.713} C_VEL
LIN {X 0,Y 312.661,Z 230.538,A -85,B 0,C 180,E1 -15670.359,E2 -15670.359} C_VEL
LIN {X 0,Y 312.646,Z 230.539,A -85,B 0,C 180,E1 -15674.875,E2 -15674.875} C_VEL
LIN {X 0,Y 312.603,Z 230.54,A -85,B 0,C 180,E1 -15679.24,E2 -15679.24} C_VEL
LIN {X 0,Y 312.567,Z 230.549,A -85,B 0,C 180,E1 -15682.814,E2 -15682.814} C_VEL
LIN {X 0,Y 312.524,Z 230.555,A -85,B 0,C 180,E1 -15686.728,E2 -15686.728} C_VEL
LIN {X 0,Y 312.515,Z 230.554,A -85,B 0,C 180,E1 -15689.653,E2 -15689.653} C_VEL
LIN {X 0,Y 312.492,Z 230.557,A -85,B 0,C 180,E1 -15693.691,E2 -15693.691} C_VEL
LIN {X 0,Y 312.514,Z 230.552,A -85,B 0,C 180,E1 -15697.386,E2 -15697.386} C_VEL
LIN {X 0,Y 312.502,Z 230.554,A -85,B 0,C 180,E1 -15700.707,E2 -15700.707} C_VEL
LIN {X 0,Y 312.503,Z 230.559,A -85,B 0,C 180,E1 -15704.2,E2 -15704.2} C_VEL
LIN {X 0,Y 312.486,Z 230.562,A -85,B 0,C 180,E1 -15707.918,E2 -15707.918} C_VEL
LIN {X 0,Y 312.519,Z 230.559,A -85,B 0,C 180,E1 -15711.913,E2 -15711.913} C_VEL
LIN {X 0,Y 312.492,Z 230.56,A -85,B 0,C 180,E1 -15715.793,E2 -15715.793} C_VEL
LIN {X 0,Y 312.511,Z 230.553,A -85,B 0,C 180,E1 -15718.857,E2 -15718.857} C_VEL
LIN {X 0,Y 312.573,Z 230.551,A -85,B 0,C 180,E1 -15721.828,E2 -15721.828} C_VEL
LIN {X 0,Y 312.577,Z 230.546,A -85,B 0,C 180,E1 -15724.713,E2 -15724.713} C_VEL
LIN {X 0,Y 312.58,Z 230.55,A -85,B 0,C 180,E1 -15727.531,E2 -15727.531} C_VEL
LIN {X 0,Y 312.633,Z 230.543,A -85,B 0,C 180,E1 -15731.658,E2 -15731.658} C_VEL
LIN {X 0,Y 312.69,Z 230.536,A -85,B 0,C 180,E1 -15735.688,E2 -15735.688} C_VEL
LIN {X 0,Y 312.698,Z 230.533,A -85,B 0,C 180,E1 -15739.643,E2 -15739.643} C_VEL
LIN {X 0,Y 312.863,Z 230.51,A -85,B 0,C 180,E1 -15742.255,E2 -15742.255} C_VEL
LIN {X 0,Y 312.713,Z 230.531,A -85,B 0,C 180,E1 -15744.843,E2 -15744.843} C_VEL
LIN {X 0,Y 312.989,Z 230.496,A -85,B 0,C 180,E1 -15748.714,E2 -15748.714} C_VEL
LIN {X 0,Y 312.987,Z 230.499,A -85,B 0,C 180,E1 -15751.287,E2 -15751.287} C_VEL
LIN {X 0,Y 312.712,Z 230.534,A -85,B 0,C 180,E1 -15755.157,E2 -15755.157} C_VEL
LIN {X 0,Y 312.856,Z 230.512,A -85,B 0,C 180,E1 -15757.745,E2 -15757.745} C_VEL
LIN {X 0,Y 312.666,Z 230.536,A -85,B 0,C 180,E1 -15761.67,E2 -15761.67} C_VEL
LIN {X 0,Y 312.696,Z 230.537,A -85,B 0,C 180,E1 -15764.886,E2 -15764.886} C_VEL
LIN {X 0,Y 312.603,Z 230.545,A -85,B 0,C 180,E1 -15769.223,E2 -15769.223} C_VEL
LIN {X 0,Y 312.542,Z 230.556,A -85,B 0,C 180,E1 -15772.788,E2 -15772.788} C_VEL
LIN {X 0,Y 312.615,Z 230.716,A -85,B 0,C 180,E1 -15775.017,E2 -15775.017} C_VEL
LIN {X 0,Y 312.997,Z 232.576,A -85,B 0,C 180,E1 -15775.605,E2 -15775.605} C_VEL
LIN {X 0,Y 321.35,Z 256.801,A -85,B 0,C 180,E1 -15776.809,E2 -15776.809} C_VEL
LIN {X 0,Y 322.134,Z 262.203,A -85,B 0,C 180,E1 -15777.001,E2 -15777.001} C_VEL
LIN {X 0,Y 319.877,Z 340.762,A -85,B 0,C 180,E1 -15778.992,E2 -15778.992} C_VEL
LIN {X 0,Y 319.189,Z 354.484,A -85,B 0,C 180,E1 -15779.603,E2 -15779.603} C_VEL
LIN {X 0,Y 318.506,Z 366.718,A -85,B 0,C 180,E1 -15780.403,E2 -15780.403} C_VEL
LIN {X 0,Y 317.471,Z 378.98,A -85,B 0,C 180,E1 -15781.474,E2 -15781.474} C_VEL
LIN {X 0,Y 316.408,Z 390.343,A -85,B 0,C 180,E1 -15782.747,E2 -15782.747} C_VEL
LIN {X 0,Y 315.372,Z 400.148,A -85,B 0,C 180,E1 -15784.116,E2 -15784.116} C_VEL
LIN {X 0,Y 314.167,Z 410.448,A -85,B 0,C 180,E1 -15785.909,E2 -15785.909} C_VEL
LIN {X 0,Y 313.184,Z 418.82,A -85,B 0,C 180,E1 -15787.718,E2 -15787.718} C_VEL
LIN {X 0,Y 312.372,Z 425.63,A -85,B 0,C 180,E1 -15789.539,E2 -15789.539} C_VEL
LIN {X 0,Y 311.769,Z 431.099,A -85,B 0,C 180,E1 -15791.35,E2 -15791.35} C_VEL
LIN {X 0,Y 311.246,Z 436.614,A -85,B 0,C 180,E1 -15793.734,E2 -15793.734} C_VEL
LIN {X 0,Y 310.784,Z 440.812,A -85,B 0,C 180,E1 -15796.349,E2 -15796.349} C_VEL
LIN {X 0,Y 310.64,Z 442.763,A -85,B 0,C 180,E1 -15798.29,E2 -15798.29} C_VEL
LIN {X 0,Y 310.627,Z 443.864,A -85,B 0,C 180,E1 -15800.691,E2 -15800.691} C_VEL
LIN {X 0,Y 310.713,Z 443.838,A -85,B 0,C 180,E1 -15802.36,E2 -15802.36} C_VEL
LIN {X 0,Y 311.085,Z 442.423,A -85,B 0,C 180,E1 -15804.895,E2 -15804.895} C_VEL
LIN {X 0,Y 311.681,Z 439.792,A -85,B 0,C 180,E1 -15807.237,E2 -15807.237} C_VEL
LIN {X 0,Y 312.646,Z 435.536,A -85,B 0,C 180,E1 -15809.617,E2 -15809.617} C_VEL
LIN {X 0,Y 312.916,Z 434.042,A -85,B 0,C 180,E1 -15810.292,E2 -15810.292} C_VEL
LIN {X 0,Y 312.743,Z 431.782,A -85,B 0,C 180,E1 -15811.293,E2 -15811.293} C_VEL
LIN {X 0,Y 310.876,Z 427.756,A -85,B 0,C 180,E1 -15812.924,E2 -15812.924} C_VEL
LIN {X 0,Y 309.15,Z 423.039,A -85,B 0,C 180,E1 -15814.504,E2 -15814.504} C_VEL
LIN {X 0,Y 309.189,Z 419.694,A -85,B 0,C 180,E1 -15815.406,E2 -15815.406} C_VEL
LIN {X 0,Y 310.951,Z 410.63,A -85,B 0,C 180,E1 -15817.405,E2 -15817.405} C_VEL
LIN {X 0,Y 312.721,Z 400.967,A -85,B 0,C 180,E1 -15819.095,E2 -15819.095} C_VEL
LIN {X 0,Y 314.545,Z 390.191,A -85,B 0,C 180,E1 -15820.589,E2 -15820.589} C_VEL
LIN {X 0,Y 316.28,Z 378.429,A -85,B 0,C 180,E1 -15821.875,E2 -15821.875} C_VEL
LIN {X 0,Y 317.702,Z 365.916,A -85,B 0,C 180,E1 -15822.924,E2 -15822.924} C_VEL
LIN {X 0,Y 318.861,Z 353.025,A -85,B 0,C 180,E1 -15823.72,E2 -15823.72} C_VEL
LIN {X 0,Y 319.595,Z 340.219,A -85,B 0,C 180,E1 -15824.25,E2 -15824.25} C_VEL
LIN {X 0,Y 322.543,Z 267.331,A -85,B 0,C 180,E1 -15826.203,E2 -15826.203} C_VEL
LIN {X 0,Y 317.177,Z 255.04,A -85,B 0,C 180,E1 -15827.248,E2 -15827.248} C_VEL
LIN {X 0,Y 310.725,Z 242.432,A -85,B 0,C 180,E1 -15828.528,E2 -15828.528} C_VEL
LIN {X 0,Y 306.699,Z 235.255,A -85,B 0,C 180,E1 -15829.362,E2 -15829.362} C_VEL
LIN {X 0,Y 305.675,Z 231.414,A -85,B 0,C 180,E1 -15830.868,E2 -15830.868} C_VEL
LIN {X 0,Y 305.805,Z 231.393,A -85,B 0,C 180,E1 -15833.402,E2 -15833.402} C_VEL
LIN {X 0,Y 305.917,Z 231.377,A -85,B 0,C 180,E1 -15838.684,E2 -15838.684} C_VEL
LIN {X 0,Y 305.916,Z 231.377,A -85,B 0,C 180,E1 -15841.317,E2 -15841.317} C_VEL
LIN {X 0,Y 305.639,Z 231.41,A -85,B 0,C 180,E1 -15845.278,E2 -15845.278} C_VEL
LIN {X 0,Y 305.751,Z 231.397,A -85,B 0,C 180,E1 -15847.928,E2 -15847.928} C_VEL
LIN {X 0,Y 305.568,Z 231.418,A -85,B 0,C 180,E1 -15851.947,E2 -15851.947} C_VEL
LIN {X 0,Y 305.576,Z 231.418,A -85,B 0,C 180,E1 -15855.015,E2 -15855.015} C_VEL
LIN {X 0,Y 305.487,Z 231.434,A -85,B 0,C 180,E1 -15858.789,E2 -15858.789} C_VEL
LIN {X 0,Y 305.459,Z 231.43,A -85,B 0,C 180,E1 -15863.042,E2 -15863.042} C_VEL
LIN {X 0,Y 305.487,Z 231.428,A -85,B 0,C 180,E1 -15866.217,E2 -15866.217} C_VEL
LIN {X 0,Y 305.441,Z 231.433,A -85,B 0,C 180,E1 -15869.043,E2 -15869.043} C_VEL
LIN {X 0,Y 305.411,Z 231.439,A -85,B 0,C 180,E1 -15871.956,E2 -15871.956} C_VEL
LIN {X 0,Y 305.438,Z 231.432,A -85,B 0,C 180,E1 -15875.117,E2 -15875.117} C_VEL
LIN {X 0,Y 305.418,Z 231.438,A -85,B 0,C 180,E1 -15878.529,E2 -15878.529} C_VEL
LIN {X 0,Y 305.436,Z 231.435,A -85,B 0,C 180,E1 -15882.589,E2 -15882.589} C_VEL
LIN {X 0,Y 305.407,Z 231.442,A -85,B 0,C 180,E1 -15886.348,E2 -15886.348} C_VEL
LIN {X 0,Y 305.445,Z 231.435,A -85,B 0,C 180,E1 -15889.896,E2 -15889.896} C_VEL
LIN {X 0,Y 305.484,Z 231.526,A -85,B 0,C 180,E1 -15893.061,E2 -15893.061} C_VEL
LIN {X 0,Y 307.614,Z 239.066,A -85,B 0,C 180,E1 -15895.783,E2 -15895.783} C_VEL
LIN {X 0,Y 310.163,Z 249.12,A -85,B 0,C 180,E1 -15899.13,E2 -15899.13} C_VEL
LIN {X 0,Y 311.742,Z 256.638,A -85,B 0,C 180,E1 -15901.405,E2 -15901.405} C_VEL
LIN {X 0,Y 314.454,Z 263.35,A -85,B 0,C 180,E1 -15901.987,E2 -15901.987} C_VEL
LIN {X 0,Y 317.967,Z 280.821,A -85,B 0,C 180,E1 -15902.998,E2 -15902.998} C_VEL
LIN {X 0,Y 320.903,Z 300.141,A -85,B 0,C 180,E1 -15903.948,E2 -15903.948} C_VEL
LIN {X 0,Y 321.289,Z 305.606,A -85,B 0,C 180,E1 -15904.162,E2 -15904.162} C_VEL
LIN {X 0,Y 318.746,Z 367.776,A -85,B 0,C 180,E1 -15905.843,E2 -15905.843} C_VEL
